// TwinCAT 3 PLC project PLC_ForTwinSAFEinTc3
// ProgramVersion: 3.1.4024.0
// libraries:
//   Tc2_EtherCAT,3.3.0.0,Beckhoff Automation GmbH
//   Tc2_MC2,3.3.2.0,Beckhoff Automation GmbH
//   Tc2_MC2_Drive,3.3.0.0,Beckhoff Automation GmbH
//   Tc2_MDP,3.3.0.0,Beckhoff Automation GmbH
//   Tc2_Standard,3.3.0.0,Beckhoff Automation GmbH
//   Tc2_System,3.3.2.0,Beckhoff Automation GmbH
//   Tc2_Utilities,3.3.1.0,Beckhoff Automation GmbH
//   Tc3_Interfaces,3.3.0.0,Beckhoff Automation GmbH
//   Tc3_Module,3.3.2.0,Beckhoff Automation GmbH
// project tree:
//   DUTs/MDP/ ST_MDP_CPU.TcDUT, ST_MDP_DiskMngmntTBL4.TcDUT, ST_MDP_DiskMngmntTBL3.TcDUT, ST_MDP_DiskMngmntTBL2.TcDUT, ST_MDP_MainboardTBL1.TcDUT, ST_MDP_DiskMngmntTBL1.TcDUT, ST_MDP_TimeTBL1.TcDUT, ST_MDP_MainboardTBL2.TcDUT (not stored), ST_MDP_MainboardTBL3.TcDUT, ST_MDP_MainboardTBL4.TcDUT, ST_MDP_NIC_Properties.TcDUT, ST_MDP_MemoryTBL1.TcDUT, ST_MDP_TimeTBL2.TcDUT
//   DUTs/Safety/ DUT_ST_InfoData.TcDUT (not stored), DUT_ST_InfoDataConnectionIn.TcDUT, DUT_ST_InfoDataConnectionOut.TcDUT, DUT_ST_InfoDataFB.TcDUT
//   / GlobalImagePool.TcGIPO (not stored), GlobalTextList.TcGTLO, PlcTask.TcTTO (not stored), Visualization Manager.TcVMO (not stored)
//   GVLs/ GVL_HMI.TcGVL, GVL_IO.TcGVL
//   POUs/Control_System_Diagnostics/ EtherCAT_Diag.TcPOU, System_Functions.TcPOU
//   POUs/ MAIN.TcPOU
//   POUs/MDP_Function_Blocks/ FB_MDP_CPU_Read.TcPOU, FB_MDP_DiskMngmnt_ReadTBL2.TcPOU, FB_MDP_DiskMngmnt_ReadTBL3.TcPOU, FB_MDP_DiskMngmnt_ReadTBL4.TcPOU, FB_MDP_Mainboard_ReadTBL1.TcPOU (not stored), FB_MDP_DiskMngmnt_ReadTBL1.TcPOU, FB_MDP_Time_ReadTBL1.TcPOU, FB_MDP_Mainboard_ReadTBL2.TcPOU, FB_MDP_Mainboard_ReadTBL3.TcPOU, FB_MDP_Mainboard_ReadTBL4.TcPOU, FB_MDP_NIC_Read.TcPOU (not stored), FB_MDP_Memory_ReadTBL1.TcPOU, FB_MDP_Time_ReadTBL2.TcPOU
//   POUs/Safety_Diagnostics/ AX5805_ADS_Reads.TcPOU, EL1904_ADS_Reads.TcPOU (not stored), EL2904_ADS_Reads.TcPOU (not stored), EL6900_ADS_Reads.TcPOU (not stored), EL6930_ADS_Reads.TcPOU, EP1908_ADS_Reads.TcPOU
//   POUs/TwinSAFE_Function_Blocks_Info/ FB_InfoAND.TcPOU (not stored), FB_InfoConnectionIn.TcPOU (not stored), FB_InfoConnectionOut.TcPOU (not stored), FB_InfoConnectionShutdown.TcPOU (not stored), FB_InfoDecoupler.TcPOU, FB_InfoEDM.TcPOU (not stored), FB_InfoEStop.TcPOU, FB_InfoMON.TcPOU, FB_InfoMuting.TcPOU, FB_InfoOperationMode.TcPOU, FB_InfoOR.TcPOU (not stored), FB_InfoRS.TcPOU, FB_InfoSafetyGroup.TcPOU, FB_InfoSR.TcPOU, FB_InfoTOF.TcPOU, FB_InfoTON.TcPOU (not stored), FB_InfoTwoHand.TcPOU (not stored)
//   VISUs/ AX5805_Specific_Diagnostics.TcVIS, AX5805_Specific_Diagnostics.TcVIS, AX5805_Specific_Diagnostics.TcVIS, EL1904_Specific_Diagnostics.TcVIS (not stored), EL1904_Specific_Diagnostics.TcVIS (not stored), EL1904_Specific_Diagnostics.TcVIS (not stored), EL2904_Specific_Diagnostics.TcVIS, EL2904_Specific_Diagnostics.TcVIS, EL2904_Specific_Diagnostics.TcVIS, EL2904_Specific_Diagnostics.TcVIS, EL6900_Specific_Diagnostics.TcVIS, EL6930_Specific_Diagnostics.TcVIS, EP1908_Specific_Diagnostics.TcVIS, EP1908_Specific_Diagnostics.TcVIS, EP1908_Specific_Diagnostics.TcVIS, EP1908_Specific_Diagnostics.TcVIS, EP6900_Specific_Diagnostics.TcVIS (not stored), EP6900_Specific_Diagnostics.TcVIS (not stored), EP6930_Specific_Diagnostics.TcVIS (not stored), EP6930_Specific_Diagnostics.TcVIS (not stored), EtherCAT_Diag1.TcVIS, EtherCAT_Diag1.TcVIS, EtherCAT_Diag1.TcVIS, EtherCAT_Diag2.TcVIS, EtherCAT_Diag2.TcVIS, EtherCAT_Diag2.TcVIS, MDP_MainboardCPUMemory.TcVIS, MDP_NicTime.TcVIS, TwinCAT_INFO.TcVIS, TwinCAT_INFO.TcVIS, TwinCAT_INFO.TcVIS, TwinSAFE.TcVIS, TwinSAFE.TcVIS, TwinSAFE.TcVIS
// real-time tasks:
//   TASK PlcTask: cycle T#1ms, priority 20, ADS port 350
// motion (NC):
//   TASK NC-Task 1 SAF: cycle T#2ms, priority 4, ADS port 501
//   TASK NC-Task 1 SVB: cycle T#10ms, priority 8, ADS port 511
//   AXIS Axis 3 (id 3)
//     OtherSettings: AllowMotionCmdToSlave=true
//     encoder EncId=1, EncType=19
//       EncPara: MaxCount=#xffffffff
//     drive DrvId=1, DrvType=16
//       DrvPara: MaxCount=#xffffffff
//         TimeComp: TaskDelayCycles=1
//     controller CtrId=1, CtrType=1
//       CtrPara: PriorControlFactor=1
//         Observer: BandWidth=20
//   AXIS Axis 4 (id 4)
//     OtherSettings: AllowMotionCmdToSlave=true
//     encoder EncId=2, EncType=19
//       EncPara: MaxCount=#xffffffff
//     drive DrvId=2, DrvType=16
//       DrvPara: MaxCount=#xffffffff
//         TimeComp: TaskDelayCycles=1
//     controller CtrId=2, CtrType=1
//       CtrPara: PriorControlFactor=1
//         Observer: BandWidth=20
// I/O:
//   DEVICE Device 1 (EtherCAT) (disabled), AmsNetId 10.12.160.29.2.1
//     Term 1 (EK1200) [EK1200-5000 EtherCAT Power supply (2A E-Bus)]
//       Term 2 (EL2004) [EL2004 4Ch. Dig. Output 24V, 0.5A]
//       Term 3 (EL1904) [EL1904, 4 Ch. Safety Input 24V, TwinSAFE]
//         modules: Module 1 (FSOES)
//       Term 4 (EL2904) [EL2904, 4 Ch. Safety Output 24V, 0.5A, TwinSAFE]
//         modules: Module 1 (FSOES), Module 2 (DO)
//       Term 5 (EL6900) [EL6900, TwinSAFE PLC]
//       Term 6 (EL1008) [EL1008 8Ch. Dig. Input 24V, 3ms]
//       Term 7 (EL2008) [EL2008 8Ch. Dig. Output 24V, 0.5A]
//       Term 8 (EL3002) [EL3002 2Ch. Ana. Input +/-10V]
//       Term 15 (EL4032) [EL4032 2Ch. Ana. Output +/-10V, 12bit]
//       Term 11 (EL7201) [EL7201 1Ch. MDP742 Servo motor output stage (50V, 4A)]
//       Term 12 (EL7201) [EL7201 1Ch. MDP742 Servo motor output stage (50V, 4A)]
//       Term 13 (EL9570) [EL9570 Buffer capacitor terminal]
//       Term 14 (EK1122) [EK1122 2 port EtherCAT junction]
//       Term 10 (EL9011) [EL9011 End Terminal]
// variable links:
//   Device 1 (EtherCAT) <-> Device 1 (EtherCAT)/Term 1 (EK1200)/Term 3 (EL1904)
//     Term 1 (EK1200)/Term 5 (EL6900)/ConnectionOutputs/Message_21 RxPDO <-> Module 1 (FSOES)/TxPDO/FSOE
//     Term 1 (EK1200)/Term 5 (EL6900)/ConnectionInputs/Message_21 TxPDO <-> Module 1 (FSOES)/RxPDO/FSOE
//   Device 1 (EtherCAT) <-> Device 1 (EtherCAT)/Term 1 (EK1200)/Term 4 (EL2904)
//     Term 1 (EK1200)/Term 5 (EL6900)/ConnectionInputs/Message_22 TxPDO <-> Module 1 (FSOES)/RxPDO/FSOE
//   Device 1 (EtherCAT) <-> Device 1 (EtherCAT)/Term 1 (EK1200)/Term 5 (EL6900)
//     Term 1 (EK1200)/Term 4 (EL2904)/Module 1 (FSOES)/TxPDO/FSOE <-> ConnectionOutputs/Message_22 RxPDO
//   NC-Task 1 SAF/Axes/Axis 3 <-> Device 1 (EtherCAT)/Term 1 (EK1200)/Term 11 (EL7201)
//     Enc/Inputs/In/nDataIn1 <-> FB Position/Position
//     Drive/Inputs/In/nState1 <-> DRV Statusword/Statusword
//     Enc/Inputs/In/nDcInputTime <-> InfoData/DcInputShift
//     Drive/Inputs/In/nDcOutputTime <-> InfoData/DcOutputShift
//     Drive/Outputs/Out/nCtrl1 <-> DRV Controlword/Controlword
//     Drive/Outputs/Out/nDataOut2 <-> DRV Target velocity/Target velocity
//     Drive/Inputs/In/nState2 <-> DRV Statusword/Statusword @bit 8
//     Drive/Outputs/Out/nCtrl2 <-> DRV Controlword/Controlword @bit 8
//   NC-Task 1 SAF/Axes/Axis 4 <-> Device 1 (EtherCAT)/Term 1 (EK1200)/Term 12 (EL7201)
//     Drive/Outputs/Out/nDataOut2 <-> DRV Target velocity/Target velocity
//     Drive/Outputs/Out/nCtrl2 <-> DRV Controlword/Controlword @bit 8
//     Enc/Inputs/In/nDcInputTime <-> InfoData/DcInputShift
//     Enc/Inputs/In/nDataIn1 <-> FB Position/Position
//     Drive/Inputs/In/nState1 <-> DRV Statusword/Statusword
//     Drive/Inputs/In/nState2 <-> DRV Statusword/Statusword @bit 8
//     Drive/Inputs/In/nDcOutputTime <-> InfoData/DcOutputShift
//     Drive/Outputs/Out/nCtrl1 <-> DRV Controlword/Controlword
//   PLC_ForTwinSAFEinTc3/PLC_ForTwinSAFEinTc3 Instance <-> Device 1 (EtherCAT)
//     PlcTask Inputs/GVL_IO.g_wStateMaster <-> Inputs/DevState
//   PLC_ForTwinSAFEinTc3/PLC_ForTwinSAFEinTc3 Instance <-> Device 1 (EtherCAT)/Term 1 (EK1200)/Term 11 (EL7201)
//     PlcTask Inputs/GVL_IO.g_stEL7201_1EcSlaveState <-> InfoData/State
//     PlcTask Inputs/GVL_IO.g_wStateEL7201_1 <-> InfoData/State
//   PLC_ForTwinSAFEinTc3/PLC_ForTwinSAFEinTc3 Instance <-> Device 1 (EtherCAT)/Term 1 (EK1200)/Term 12 (EL7201)
//     PlcTask Inputs/GVL_IO.g_stEL7201_2EcSlaveState <-> InfoData/State
//     PlcTask Inputs/GVL_IO.g_wStateEL7201_2 <-> InfoData/State
//   PLC_ForTwinSAFEinTc3/PLC_ForTwinSAFEinTc3 Instance <-> Device 1 (EtherCAT)/Term 1 (EK1200)/Term 14 (EK1122)
//     PlcTask Inputs/GVL_IO.g_stEK1122_EcSlaveState <-> InfoData/State
//     PlcTask Inputs/GVL_IO.g_wStateEK1122 <-> InfoData/State
//   PLC_ForTwinSAFEinTc3/PLC_ForTwinSAFEinTc3 Instance <-> Device 1 (EtherCAT)/Term 1 (EK1200)/Term 15 (EL4032)
//     PlcTask Inputs/GVL_IO.g_stEL4032EcSlaveState <-> InfoData/State
//     PlcTask Inputs/GVL_IO.g_wStateEL4032 <-> InfoData/State
//   PLC_ForTwinSAFEinTc3/PLC_ForTwinSAFEinTc3 Instance <-> Device 1 (EtherCAT)/Term 1 (EK1200)/Term 2 (EL2004)
//     PlcTask Outputs/GVL_IO.g_xOutput1 <-> Channel 1/Output
//     PlcTask Inputs/GVL_IO.g_wStateEL2004 <-> InfoData/State
//     PlcTask Inputs/GVL_IO.g_stEL2004EcSlaveState <-> InfoData/State
//   PLC_ForTwinSAFEinTc3/PLC_ForTwinSAFEinTc3 Instance <-> Device 1 (EtherCAT)/Term 1 (EK1200)/Term 3 (EL1904)
//     PlcTask Inputs/GVL_IO.g_stEL1904EcSlaveState <-> InfoData/State
//     PlcTask Inputs/GVL_IO.g_wStateEL1904 <-> InfoData/State
//   PLC_ForTwinSAFEinTc3/PLC_ForTwinSAFEinTc3 Instance <-> Device 1 (EtherCAT)/Term 1 (EK1200)/Term 4 (EL2904)
//     PlcTask Inputs/GVL_IO.g_wStateEL2904 <-> InfoData/State
//     PlcTask Inputs/GVL_IO.g_stEL2904EcSlaveState <-> InfoData/State
//   PLC_ForTwinSAFEinTc3/PLC_ForTwinSAFEinTc3 Instance <-> Device 1 (EtherCAT)/Term 1 (EK1200)/Term 5 (EL6900)
//     PlcTask Inputs/GVL_IO.g_xTS_SafetyGroup1_COMerror <-> StandardInputs/Standard Out Var 2
//     PlcTask Outputs/GVL_IO.g_xTS_ErrAck <-> StandardOutputs/Standard In Var 1
//     PlcTask Inputs/GVL_IO.g_xTS_SafetyGroup1_FBerror <-> StandardInputs/Standard Out Var 3
//     PlcTask Inputs/GVL_IO.g_xTS_EDM_Error <-> StandardInputs/Standard Out Var 9
//     PlcTask Inputs/GVL_IO.g_stEL6900EcSlaveState <-> InfoData/State
//     PlcTask Inputs/GVL_IO.g_xTS_EStop_Error <-> StandardInputs/Standard Out Var 5
//     PlcTask Inputs/GVL_IO.g_uiTS_ProjectCRC <-> Device Info Data/Project CRC
//     PlcTask Inputs/GVL_IO.g_stTS_InfoGroup1/usiMapDiag <-> TwinSAFE Group Info Data/TwinSafeGroup1 Info Data/Diag
//     PlcTask Inputs/GVL_IO.g_stTS_InfoConnection1/usiMapState <-> Connection Info Data/Message_21 Info Data/State
//     PlcTask Inputs/GVL_IO.g_stTS_InfoConnection2/usiMapState <-> Connection Info Data/Message_22 Info Data/State
//     PlcTask Inputs/GVL_IO.g_stTS_InfoAND1/uiMapDiag <-> Function Block Info Data/TwinSafeGroup1.Network1.FBAnd1 Info Data/Diag
//     PlcTask Inputs/GVL_IO.g_stTS_InfoAND2/uiMapDiag <-> Function Block Info Data/TwinSafeGroup1.Network1.FBAnd2 Info Data/Diag
//     PlcTask Inputs/GVL_IO.g_stTS_InfoConnection1/byInputSignals <-> Connection Info Data/Message_21 Info Data/Input Safe Data Byte 0
//     PlcTask Inputs/GVL_IO.g_wStateEL6900 <-> InfoData/State
//     PlcTask Inputs/GVL_IO.g_stTS_InfoEStop1/uiMapDiag <-> Function Block Info Data/TwinSafeGroup1.Network1.FBEstop1 Info Data/Diag
//     PlcTask Inputs/GVL_IO.g_stTS_InfoConnection2/byOutputSignals <-> Connection Info Data/Message_22 Info Data/Output Safe Data Byte 0
//     PlcTask Inputs/GVL_IO.g_stTS_InfoEDM/uiMapDiag <-> Function Block Info Data/TwinSafeGroup1.Network1.FBEdm1 Info Data/Diag
//     PlcTask Inputs/GVL_IO.g_stTS_InfoAND1/usiMapState <-> Function Block Info Data/TwinSafeGroup1.Network1.FBAnd1 Info Data/State
//     PlcTask Inputs/GVL_IO.g_stTS_InfoAND2/usiMapState <-> Function Block Info Data/TwinSafeGroup1.Network1.FBAnd2 Info Data/State
//     PlcTask Inputs/GVL_IO.g_stTS_InfoTON/uiMapDiag <-> Function Block Info Data/TwinSafeGroup1.Network1.FBTon1 Info Data/Diag
//     PlcTask Inputs/GVL_IO.g_udiTS_SerialNumber <-> Device Info Data/Serial Number
//     PlcTask Inputs/GVL_IO.g_stTS_InfoTOF/uiMapDiag <-> Function Block Info Data/TwinSafeGroup1.Network1.FBTof1 Info Data/Diag
//     PlcTask Inputs/GVL_IO.g_stTS_InfoConnection1/usiMapDiag <-> Connection Info Data/Message_21 Info Data/Diag
//     PlcTask Inputs/GVL_IO.g_stTS_InfoConnection2/usiMapDiag <-> Connection Info Data/Message_22 Info Data/Diag
//     PlcTask Inputs/GVL_IO.g_stTS_InfoTOF/usiMapState <-> Function Block Info Data/TwinSafeGroup1.Network1.FBTof1 Info Data/State
//     PlcTask Inputs/GVL_IO.g_xTS_EStop_OFF_Delay_Complete <-> StandardInputs/Standard Out Var 8
//     PlcTask Inputs/GVL_IO.g_xTS_EStop_Complete <-> StandardInputs/Standard Out Var 6
//     PlcTask Outputs/GVL_IO.g_xTS_EStop_Reset <-> StandardOutputs/Standard In Var 12
//     PlcTask Inputs/GVL_IO.g_xTS_EStop_ON_Delay_Complete <-> StandardInputs/Standard Out Var 7
//     PlcTask Inputs/GVL_IO.g_stTS_InfoGroup1/usiMapState <-> TwinSAFE Group Info Data/TwinSafeGroup1 Info Data/State
//     PlcTask Inputs/GVL_IO.g_stTS_InfoEStop1/usiMapState <-> Function Block Info Data/TwinSafeGroup1.Network1.FBEstop1 Info Data/State
//     PlcTask Inputs/GVL_IO.g_stTS_InfoEDM/usiMapState <-> Function Block Info Data/TwinSafeGroup1.Network1.FBEdm1 Info Data/State
//     PlcTask Inputs/GVL_IO.g_stTS_InfoTON/usiMapState <-> Function Block Info Data/TwinSafeGroup1.Network1.FBTon1 Info Data/State
//   PLC_ForTwinSAFEinTc3/PLC_ForTwinSAFEinTc3 Instance <-> Device 1 (EtherCAT)/Term 1 (EK1200)/Term 6 (EL1008)
//     PlcTask Inputs/GVL_IO.g_wStateEL1008 <-> InfoData/State
//     PlcTask Inputs/GVL_IO.g_stEL1008EcSlaveState <-> InfoData/State
//   PLC_ForTwinSAFEinTc3/PLC_ForTwinSAFEinTc3 Instance <-> Device 1 (EtherCAT)/Term 1 (EK1200)/Term 7 (EL2008)
//     PlcTask Inputs/GVL_IO.g_stEL2008EcSlaveState <-> InfoData/State
//     PlcTask Inputs/GVL_IO.g_wStateEL2008 <-> InfoData/State
//   PLC_ForTwinSAFEinTc3/PLC_ForTwinSAFEinTc3 Instance <-> Device 1 (EtherCAT)/Term 1 (EK1200)/Term 8 (EL3002)
//     PlcTask Inputs/GVL_IO.g_wStateEL3002 <-> InfoData/State
//     PlcTask Inputs/GVL_IO.g_stEL3002EcSlaveState <-> InfoData/State

// ---- DUTs/MDP/ST_MDP_CPU.TcDUT
TYPE ST_MDP_CPU :
STRUCT
	uiLen			:UINT;			// Length
	udiCPUfrequency	:UDINT;			// CPU Frequency in MHz
	uiCPUusage		:UINT;			// Current CPU Usage [%]
	iCPUtemp 		:INT;			// Current CPU temperature in DegC
END_STRUCT
END_TYPE

// ---- DUTs/MDP/ST_MDP_DiskMngmntTBL4.TcDUT
TYPE ST_MDP_DiskMngmntTBL4 :
STRUCT
	uiLen				:UINT;	// Length
	udiDriveType1		:UDINT;	// DRV_UNKNOWN = 0, DRV_FIXED = 1, DRV_REMOVABLE = 2, DRV_CDROM = 4 
	udiDriveType2		:UDINT;	// DRV_UNKNOWN = 0, DRV_FIXED = 1, DRV_REMOVABLE = 2, DRV_CDROM = 4 
	udiDriveType3		:UDINT;	// DRV_UNKNOWN = 0, DRV_FIXED = 1, DRV_REMOVABLE = 2, DRV_CDROM = 4 
	udiDriveType4		:UDINT;	// DRV_UNKNOWN = 0, DRV_FIXED = 1, DRV_REMOVABLE = 2, DRV_CDROM = 4 
	udiDriveType5		:UDINT;	// DRV_UNKNOWN = 0, DRV_FIXED = 1, DRV_REMOVABLE = 2, DRV_CDROM = 4 
	udiDriveType6		:UDINT;	// DRV_UNKNOWN = 0, DRV_FIXED = 1, DRV_REMOVABLE = 2, DRV_CDROM = 4 
END_STRUCT
END_TYPE

// ---- DUTs/MDP/ST_MDP_DiskMngmntTBL3.TcDUT
TYPE ST_MDP_DiskMngmntTBL3 :
STRUCT
	uiLen				:UINT;			// Length
	sFileSystemName1	:T_MaxSTRING;	// File System Name
	sFileSystemName2	:T_MaxSTRING;	// File System Name
	sFileSystemName3	:T_MaxSTRING;	// File System Name
	sFileSystemName4	:T_MaxSTRING;	// File System Name
	sFileSystemName5	:T_MaxSTRING;	// File System Name
	sFileSystemName6	:T_MaxSTRING;	// File System Name
END_STRUCT
END_TYPE

// ---- DUTs/MDP/ST_MDP_DiskMngmntTBL2.TcDUT
TYPE ST_MDP_DiskMngmntTBL2 :
STRUCT
	uiLen				:UINT;			// Length
	sVolumeLabel1		:T_MaxSTRING;	// Volume Label
	sVolumeLabel2		:T_MaxSTRING;	// Volume Label
	sVolumeLabel3		:T_MaxSTRING;	// Volume Label
	sVolumeLabel4		:T_MaxSTRING;	// Volume Label
	sVolumeLabel5		:T_MaxSTRING;	// Volume Label
	sVolumeLabel6		:T_MaxSTRING;	// Volume Label
END_STRUCT
END_TYPE

// ---- DUTs/MDP/ST_MDP_MainboardTBL1.TcDUT
TYPE ST_MDP_MainboardTBL1 :
STRUCT
	uiLen					:UINT;			// Length
	sMainboardType			:T_MaxSTRING;	// CX model
	sMainboardSN			:T_MaxSTRING;	// CX Serial number
	sMainboardProdDate		:T_MaxSTRING;	// CX production date
	udiMainboardBootCount	:UDINT;			// Number of times this CX has been booted
	udiMainboardOperTime	:UDINT;			// Number of Minutes this CX has been in operation
	diMainboardMinTemp		:DINT;			// CX lowest operating temperature monitored
	diMainboardMaxTemp		:DINT;			// CX highest operating temperature monitored
	diMainboardMinVolt		:DINT;			// CX lowest input voltage monitored in mV - 5000 is Nominal value
	diMainboardMaxVolt		:DINT;			// CX highest input voltage monitored in mV - 5000 is Nominal value
	iMainboardActualTemp	:INT;			// CX current actual temperature
END_STRUCT
END_TYPE

// ---- DUTs/MDP/ST_MDP_DiskMngmntTBL1.TcDUT
TYPE ST_MDP_DiskMngmntTBL1 :
STRUCT
	uiLen				:UINT;			// Length
	sDriveLetter1		:STRING(8);		// Drive Letter
	sDriveLetter2		:STRING(8);		// Drive Letter
	sDriveLetter3		:STRING(8);		// Drive Letter
	sDriveLetter4		:STRING(8);		// Drive Letter
	sDriveLetter5		:STRING(8);		// Drive Letter
	sDriveLetter6		:STRING(8);		// Drive Letter
END_STRUCT
END_TYPE

// ---- DUTs/MDP/ST_MDP_TimeTBL1.TcDUT
TYPE ST_MDP_TimeTBL1 :
STRUCT
	uiLen					:UINT;			// Length
	sSNTP_Server			:STRING(255);	// SNTP Server
	udiSNTP_Refresh			:UDINT;			// SNTP Refresh in Seconds
	udiSec_Since_1_1_1970	:UDINT;			// Seconds since midnight January 1, 1970
	sDateTime_Presentation	:T_MaxSTRING;	// Textual DateTime presentation (ISO 8601) YYYY-MM-DDThh:mm:ss.sTZD
	uiTimezone				:UINT;			// Timezone
END_STRUCT
END_TYPE

// ---- DUTs/MDP/ST_MDP_MainboardTBL3.TcDUT
TYPE ST_MDP_MainboardTBL3 :
STRUCT
	uiLen					:UINT;				// Length *)
	sMainboard1p05v			:STRING;			// Nominal voltage of 1.05 volt in power supply - mV
	sMainboardVccCore		:STRING;			// Nominal voltage of Vcc Core in processor - mV
	sMainboard5v			:STRING;			// Nominal voltage of 5 volt in power supply - mV
	sMainboard12v			:STRING;			// Nominal voltage of 12 volt in power supply - mV
	sMainboardVBatt			:STRING;			// Nominal voltage of 3 volt Battery - mV
	sMainboardPwrCtrlVcc	:STRING;			// Nominal voltage of 5 volt in UNKNOWN - mV
	sMainboardCX2100_5v		:STRING;			// Nominal voltage of 5 volt supply in CX2100 - mV
	sMainboardCX2100_12v	:STRING;			// Nominal voltage of 12 volt supply in CX2100 - mV
	sMainboardCX2100_24v	:STRING;			// Nominal voltage of 24 volt supply in CX2100 - mV
END_STRUCT
END_TYPE

// ---- DUTs/MDP/ST_MDP_MainboardTBL4.TcDUT
TYPE ST_MDP_MainboardTBL4 :
STRUCT
	uiLen					:UINT;			// Length
	iMainboard1p05v			:INT;			// Actual voltage of 1.05 volt in power supply - mV
	iMainboardVccCore		:INT;			// Actual voltage of Vcc Core in processor - mV
	iMainboard5v			:INT;			// Actual voltage of 5 volt in power supply - mV
	iMainboard12v			:INT;			// Actual voltage of 12 volt in power supply - mV
	iMainboardVBatt			:INT;			// Actual voltage of 3 volt Battery - mV
	iMainboardPwrCtrlVcc	:INT;			// Actual voltage of 5 volt in UNKNOWN - mV
	iMainboardCX2100_5v		:INT;			// Actual voltage of 5 volt supply in CX2100 - mV
	iMainboardCX2100_12v	:INT;			// Actual voltage of 12 volt supply in CX2100 - mV
	iMainboardCX2100_24v	:INT;			// Actual voltage of 24 volt supply in CX2100 - mV
END_STRUCT
END_TYPE

// ---- DUTs/MDP/ST_MDP_NIC_Properties.TcDUT
TYPE ST_MDP_NIC_Properties :
STRUCT
	uiLen			:UINT;			// Length
	sMACAddress		:T_MaxSTRING;	// MAC Address
	sIPAddress		:T_MaxSTRING;	// IPv4 Address
	sSubnetMask		:T_MaxSTRING;	// IPv4 Subnet Mask
	xDHCP			:BOOL;			// DHCP
	iReserved		:BYTE;
	sDefaultGateway	:T_MaxSTRING;	// IPv4 Default Gateway
END_STRUCT
END_TYPE

// ---- DUTs/MDP/ST_MDP_MemoryTBL1.TcDUT
TYPE ST_MDP_MemoryTBL1 :
STRUCT
	uiLen					:UINT;			// Length
	udiProgMemAllocated		:UDINT;			// Program Memory Allocated
	udiProgMemAvailable		:UDINT;			// Program Memory Available
	udiStorageMemAllocated	:UDINT;			// Storage Memory Allocated (available for Windows CE)
	udiStorageMemAvailable	:UDINT;			// Storage Memory Available (available for Windows CE)
	udiMemoryDivision		:UDINT;			// Memory Division (available for Windows CE)
END_STRUCT
END_TYPE

// ---- DUTs/MDP/ST_MDP_TimeTBL2.TcDUT
TYPE ST_MDP_TimeTBL2 :
STRUCT
	uiLen					:UINT;			// Length
	sTimezone1				:T_MaxSTRING;	// Timezone1
	sTimezone2				:T_MaxSTRING;	// Timezone2
	sTimezone3				:T_MaxSTRING;	// Timezone3
	sTimezone4				:T_MaxSTRING;	// Timezone4
	sTimezone5				:T_MaxSTRING;	// Timezone5
	sTimezone6				:T_MaxSTRING;	// Timezone6
	sTimezone7				:T_MaxSTRING;	// Timezone7
	sTimezone8				:T_MaxSTRING;	// Timezone8
	sTimezone9				:T_MaxSTRING;	// Timezone9
	sTimezone10				:T_MaxSTRING;	// Timezone10
	sTimezone11				:T_MaxSTRING;	// Timezone11
	sTimezone12				:T_MaxSTRING;	// Timezone12
	sTimezone13				:T_MaxSTRING;	// Timezone13
	sTimezone14				:T_MaxSTRING;	// Timezone14
	sTimezone15				:T_MaxSTRING;	// Timezone15
	sTimezone16				:T_MaxSTRING;	// Timezone16
	sTimezone17				:T_MaxSTRING;	// Timezone17
	sTimezone18				:T_MaxSTRING;	// Timezone18
	sTimezone19				:T_MaxSTRING;	// Timezone19
	sTimezone20				:T_MaxSTRING;	// Timezone20
	sTimezone21				:T_MaxSTRING;	// Timezone21
	sTimezone22				:T_MaxSTRING;	// Timezone22
	sTimezone23				:T_MaxSTRING;	// Timezone23
	sTimezone24				:T_MaxSTRING;	// Timezone24
	sTimezone25				:T_MaxSTRING;	// Timezone25
	sTimezone26				:T_MaxSTRING;	// Timezone26
	sTimezone27				:T_MaxSTRING;	// Timezone27
	sTimezone28				:T_MaxSTRING;	// Timezone28
	sTimezone29				:T_MaxSTRING;	// Timezone29
	sTimezone30				:T_MaxSTRING;	// Timezone30
	sTimezone31				:T_MaxSTRING;	// Timezone31
	sTimezone32				:T_MaxSTRING;	// Timezone32
	sTimezone33				:T_MaxSTRING;	// Timezone33
	sTimezone34				:T_MaxSTRING;	// Timezone34
	sTimezone35				:T_MaxSTRING;	// Timezone35
	sTimezone36				:T_MaxSTRING;	// Timezone36
	sTimezone37				:T_MaxSTRING;	// Timezone37
	sTimezone38				:T_MaxSTRING;	// Timezone38
	sTimezone39				:T_MaxSTRING;	// Timezone39
	sTimezone40				:T_MaxSTRING;	// Timezone40
	sTimezone41				:T_MaxSTRING;	// Timezone41
	sTimezone42				:T_MaxSTRING;	// Timezone42
	sTimezone43				:T_MaxSTRING;	// Timezone43
	sTimezone44				:T_MaxSTRING;	// Timezone44
	sTimezone45				:T_MaxSTRING;	// Timezone45
	sTimezone46				:T_MaxSTRING;	// Timezone46
	sTimezone47				:T_MaxSTRING;	// Timezone47
	sTimezone48				:T_MaxSTRING;	// Timezone48
	sTimezone49				:T_MaxSTRING;	// Timezone49
	sTimezone50				:T_MaxSTRING;	// Timezone50
	sTimezone51				:T_MaxSTRING;	// Timezone51
	sTimezone52				:T_MaxSTRING;	// Timezone52
	sTimezone53				:T_MaxSTRING;	// Timezone53
	sTimezone54				:T_MaxSTRING;	// Timezone54
	sTimezone55				:T_MaxSTRING;	// Timezone55
	sTimezone56				:T_MaxSTRING;	// Timezone56
	sTimezone57				:T_MaxSTRING;	// Timezone57
	sTimezone58				:T_MaxSTRING;	// Timezone58
	sTimezone59				:T_MaxSTRING;	// Timezone59
	sTimezone60				:T_MaxSTRING;	// Timezone60
	sTimezone61				:T_MaxSTRING;	// Timezone61
	sTimezone62				:T_MaxSTRING;	// Timezone62
	sTimezone63				:T_MaxSTRING;	// Timezone63
	sTimezone64				:T_MaxSTRING;	// Timezone64
	sTimezone65				:T_MaxSTRING;	// Timezone65
	sTimezone66				:T_MaxSTRING;	// Timezone66
	sTimezone67				:T_MaxSTRING;	// Timezone67
	sTimezone68				:T_MaxSTRING;	// Timezone68
	sTimezone69				:T_MaxSTRING;	// Timezone69
	sTimezone70				:T_MaxSTRING;	// Timezone70
	sTimezone71				:T_MaxSTRING;	// Timezone71
	sTimezone72				:T_MaxSTRING;	// Timezone72
	sTimezone73				:T_MaxSTRING;	// Timezone73
	sTimezone74				:T_MaxSTRING;	// Timezone74
	sTimezone75				:T_MaxSTRING;	// Timezone75
	sTimezone76				:T_MaxSTRING;	// Timezone76
	sTimezone77				:T_MaxSTRING;	// Timezone77
	sTimezone78				:T_MaxSTRING;	// Timezone78
	sTimezone79				:T_MaxSTRING;	// Timezone79
	sTimezone80				:T_MaxSTRING;	// Timezone80
	sTimezone81				:T_MaxSTRING;	// Timezone81
	sTimezone82				:T_MaxSTRING;	// Timezone82
	sTimezone83				:T_MaxSTRING;	// Timezone83
	sTimezone84				:T_MaxSTRING;	// Timezone84
	sTimezone85				:T_MaxSTRING;	// Timezone85
	sTimezone86				:T_MaxSTRING;	// Timezone86
	sTimezone87				:T_MaxSTRING;	// Timezone87
	sTimezone88				:T_MaxSTRING;	// Timezone88
	sTimezone89				:T_MaxSTRING;	// Timezone89
	sTimezone90				:T_MaxSTRING;	// Timezone90
	sTimezone91				:T_MaxSTRING;	// Timezone91
	sTimezone92				:T_MaxSTRING;	// Timezone92
	sTimezone93				:T_MaxSTRING;	// Timezone93
	sTimezone94				:T_MaxSTRING;	// Timezone94
	sTimezone95				:T_MaxSTRING;	// Timezone95
	sTimezone96				:T_MaxSTRING;	// Timezone96
	sTimezone97				:T_MaxSTRING;	// Timezone97
	sTimezone98				:T_MaxSTRING;	// Timezone98
	sTimezone99				:T_MaxSTRING;	// Timezone99
	sTimezone100			:T_MaxSTRING;	// Timezone100
	sTimezone101			:T_MaxSTRING;	// Timezone101
END_STRUCT
END_TYPE

// ---- DUTs/Safety/DUT_ST_InfoDataConnectionIn.TcDUT
TYPE DUT_ST_InfoDataConnectionIn :
STRUCT
	// Safety input connections use this structure
	usiMapState 				: 	USINT ;
	usiMapDiag  				: 	USINT ;
	byInputSignals 				: 	BYTE ;	
END_STRUCT
END_TYPE

// ---- DUTs/Safety/DUT_ST_InfoDataConnectionOut.TcDUT
TYPE DUT_ST_InfoDataConnectionOut :
STRUCT
	///  Safety output connections use this structure
	usiMapState					: 	USINT ;
	usiMapDiag					: 	USINT ;
	byOutputSignals				: 	BYTE ;
END_STRUCT
END_TYPE

// ---- DUTs/Safety/DUT_ST_InfoDataFB.TcDUT
TYPE DUT_ST_InfoDataFB :
STRUCT
	// Safety FBs use this structure
	usiMapState 		: 	USINT ;
	uiMapDiag  			: 	UINT ;	
END_STRUCT
END_TYPE

// ---- GVLs/GVL_HMI.TcGVL
VAR_GLOBAL
//		8-2-2012
// 		This Program has been supplied by Beckhoff Automation As-Is and is intended only as an example 
//		implementation. Functionality is not guaranteed. 
//	
	// TwinSAFE project CRC	
	g_uiHMI_ProjectCRC						: 	UINT ;
	g_udiHMI_SerialNumber					: 	UDINT ;	

	// Commands to TwinSAFE controller's safety  group
	g_xHMI_ErrAckPB							: 	BOOL ;
	g_xHMI_EStopResetPB						: 	BOOL ;

	// Feedback from TwinSAFE controller's safety group
	g_xHMI_SafetyGroup1_FBerrorLT			: 	BOOL ;
	g_xHMI_SafetyGroup1_COMerrorLT			: 	BOOL ;
	
	// Feedback from TwinSAFE controller's Function Blocks
	g_xHMI_EDMerrorLT						: 	BOOL ;
	g_xHMI_EStop_CompleteLT					: 	BOOL ;
	g_xHMI_EStop_errorLT					: 	BOOL ;
	g_xHMI_EStop_OFF_Delay_CompleteLT		: 	BOOL ;
	g_xHMI_EStop_ON_Delay_CompleteLT		: 	BOOL ;
	
	// Safety Group1 Info 
	g_sHMI_StatusGroup1						: 	STRING ;
	
	// Safety Connection1 Info
	g_sHMI_StateConn1						: 	STRING ;
	g_sHMI_DiagConn1						: 	STRING ;
	g_xHMI_EL1904Ch1						: 	BOOL ;
	g_xHMI_EL1904Ch2						: 	BOOL ;
	g_xHMI_EL1904Ch3						: 	BOOL ;
	g_xHMI_EL1904Ch4						: 	BOOL ;

	// Safety Connection2 Info
	g_sHMI_StateConn2						: 	STRING ;
	g_sHMI_DiagConn2						: 	STRING ;
	g_xHMI_EL2904Ch1						: 	BOOL ;
	g_xHMI_EL2904Ch2						: 	BOOL ;
	g_xHMI_EL2904Ch3						: 	BOOL ;
	g_xHMI_EL2904Ch4						: 	BOOL ;

	// Future Safety Connection Info for EP1908-0002
	g_xHMI_EP1908Ch1						: 	BOOL ;
	g_xHMI_EP1908Ch2						: 	BOOL ;	
	g_xHMI_EP1908Ch3						: 	BOOL ;
	g_xHMI_EP1908Ch4						: 	BOOL ;
	g_xHMI_EP1908Ch5						: 	BOOL ;
	g_xHMI_EP1908Ch6						: 	BOOL ;
	g_xHMI_EP1908Ch7						: 	BOOL ;	
	g_xHMI_EP1908Ch8						: 	BOOL ;
	
	// Safety AND#1 FB Info
	g_sHMI_StatusAND1						:	STRING ;

	// Safety EStop#1 FB Info
	g_sHMI_StatusEStop1						: 	STRING ;	
	g_sHMI_DiagEStop1						: 	STRING ;	

	// Safety AND#2 FB Info
	g_sHMI_StatusAND2						: 	STRING ;

	// Safety TON FB Info
	g_sHMI_StatusTON						: 	STRING ;

	// Safety TOF FB Info
	g_sHMI_StatusTOF						: 	STRING ;

	// Safety EDM FB Info
	g_sHMI_StatusEDM						: 	STRING ;
	g_sHMI_DiagEDM							: 	STRING ;

	//ADS Read Function Block Constants
	gc_sADSNetID							: 	STRING 		:= '10.12.160.29.2.1' ;
	gc_uiEL2004_EtherCATAdr					:	UINT 		:= 1001 ;
	gc_uiEL1904_EtherCATAdr					:	UINT 		:= 1002 ;
	gc_uiEL2904_EtherCATAdr					:	UINT 		:= 1003 ;
	gc_uiEL6900_EtherCATAdr					:	UINT 		:= 1004 ;
	gc_uiEL1008_EtherCATAdr					:	UINT 		:= 1005 ;
	gc_uiEL2008_EtherCATAdr					:	UINT 		:= 1006 ;
	gc_uiEL3002_EtherCATAdr					:	UINT 		:= 1007 ;
	gc_uiEL4032_EtherCATAdr					:	UINT 		:= 1008 ;
	gc_uiEL7201_1_EtherCATAdr				:	UINT 		:= 1009 ;
	gc_uiEL7201_2_EtherCATAdr				:	UINT 		:= 1010 ;
	gc_uiEK1122_EtherCATAdr					:	UINT 		:= 1011 ;
	
	//EL1904 Safety Terminal CoE Objects of Interest(via ADS Reads)
	g_dwHMI_EL1904Sn						: 	DWORD ;  //EL1904 Serial Number
	g_wHMI_EL1904DSw						: 	WORD ;   //EL1904 DIP Switch Setting
	g_sHMI_EL1904_HWvers					: 	STRING(2) ;//EL1904 Hardware Version
	g_sHMI_EL1904_FWvers					: 	STRING(2) ;	//EL1904 Firmware Version
	g_wHMI_EL1904PriMCTemp					: 	WORD ;   //EL1904 MC1 Actual Termperature In DegC
	g_wHMI_EL1904SecMCTemp					: 	WORD ;   //EL1904 MC2 Actual Termperature In DegC
	g_wHMI_EL1904SecMC_Volts				: 	LREAL ;  //EL1904 MC1 Actual Voltage (3.3v is nominal)
	g_wHMI_EL1904PriMC_Volts				: 	LREAL ;  //EL1904 MC2 Actual Voltage (3.3v is nominal)
	g_xHMI_EL1904SenT1						: 	BOOL ;   //EL1904 Sensor Test Error on CH1
	g_xHMI_EL1904SenT2						: 	BOOL ;   //EL1904 Sensor Test Error on CH2
	g_xHMI_EL1904SenT3						: 	BOOL ;   //EL1904 Sensor Test Error on CH3
	g_xHMI_EL1904SenT4						: 	BOOL ;   //EL1904 Sensor Test Error on CH4
	g_xHMI_EL1904_2CHEval_Pair1				: 	BOOL ;   //EL1904 2CH-Eval Error Pair1 (CH1 and CH2 not same value)
	g_xHMI_EL1904_2CHEval_Pair2				: 	BOOL ;   //EL1904 2CH-Eval Error Pair2 (CH3 and CH4 not same value)
	g_xHMI_EL1904_SMiPair_Pair1				: 	BOOL ;   //EL1904 Safety Mat Error Pair1 (CH1 and CH2 not same value)
	g_xHMI_EL1904_SMiPair_Pair2				: 	BOOL ;   //EL1904 Safety Mat Error Pair2 (CH3 and CH4 not same value)
	g_xHMI_EL1904_SMExtSupply_CH1			: 	BOOL ;   //EL1904 Safety Mat Error - External Supply CH1 (CH1 test pulses missing)
	g_xHMI_EL1904_SMExtSupply_CH2			: 	BOOL ;   //EL1904 Safety Mat Error - External Supply CH2 (CH2 test pulses missing)
	g_xHMI_EL1904_SMExtSupply_CH3			: 	BOOL ;   //EL1904 Safety Mat Error - External Supply CH3 (CH3 test pulses missing)
	g_xHMI_EL1904_SMExtSupply_CH4			: 	BOOL ;   //EL1904 Safety Mat Error - External Supply CH4 (CH4 test pulses missing)
	g_xHMI_EL1904_ErrClearPB				: 	BOOL ;   //EL1904 HMI Screen Errors Clear Pushbutton
	
	//EL1904 Safety Terminal FEATURES
	g_sHMI_EL1904_OperatingMode				: 	STRING ;  //EL1904 FEATURE - Operating Mode
	g_xHMI_EL1904_SensTestActive1			: 	BOOL ;	  //EL1904 FEATURE - CH1 Sensor Test Active
	g_xHMI_EL1904_SensTestActive2			: 	BOOL ;	  //EL1904 FEATURE - CH2 Sensor Test Active
	g_xHMI_EL1904_SensTestActive3			: 	BOOL ;	  //EL1904 FEATURE - CH3 Sensor Test Active
	g_xHMI_EL1904_SensTestActive4			: 	BOOL ;	  //EL1904 FEATURE - CH4 Sensor Test Active
	g_sHMI_EL1904_LogicCh1andCh2			: 	STRING ;  //EL1904 FEATURE - CH1 and CH2 Logic
	g_sHMI_EL1904_LogicCh3andCh4			: 	STRING ;  //EL1904 FEATURE - CH3 and CH4 Logic
	
	//EL2904 Safety Terminal CoE Objects of Interest(via ADS Reads)
	g_dwHMI_EL2904Sn						:	DWORD ;  //EL2904 Serial Number
	g_wHMI_EL2904DSw						: 	WORD ;   //EL2904 DIP Switch Setting
	g_sHMI_EL2904_HWvers					: 	STRING(2) ;//EL2904 Hardware Version
	g_sHMI_EL2904_FWvers					: 	STRING(2) ;//EL2904 Firmware Version
	g_wHMI_EL2904PriMCTemp					: 	WORD ;   //EL2904 MC1 Actual Termperature In DegC
	g_wHMI_EL2904SecMCTemp					: 	WORD ;   //EL2904 MC2 Actual Termperature In DegC
	g_wHMI_EL2904SecMC_Volts				: 	LREAL ;  //EL2904 MC1 Actual Voltage (3.3v is nominal)
	g_wHMI_EL2904PriMC_Volts				: 	LREAL ;  //EL2904 MC2 Actual Voltage (3.3v is nominal)
	g_xHMI_EL2904_ExtSup_CrossCirErr_Out1	: 	BOOL ;   //EL2904 ExtSupply, Cross-Circuit (No Test Pulses) Error on CH1
	g_xHMI_EL2904_ExtSup_CrossCirErr_Out2	: 	BOOL ;   //EL2904 ExtSupply, Cross-Circuit (No Test Pulses) Error on CH2
	g_xHMI_EL2904_ExtSup_CrossCirErr_Out3	: 	BOOL ;   //EL2904 ExtSupply, Cross-Circuit (No Test Pulses) Error on CH3
	g_xHMI_EL2904_ExtSup_CrossCirErr_Out4	: 	BOOL ;   //EL2904 ExtSupply, Cross-Circuit (No Test Pulses) Error on CH4
	g_xHMI_EL2904_OutLoadErr_Out1			: 	BOOL ;   //EL2904 Open Load, I<20mA, or I>500mA on CH1
	g_xHMI_EL2904_OutLoadErr_Out2			: 	BOOL ;   //EL2904 Open Load, I<20mA, or I>500mA on CH2
	g_xHMI_EL2904_OutLoadErr_Out3			: 	BOOL ;   //EL2904 Open Load, I<20mA, or I>500mA on CH3
	g_xHMI_EL2904_OutLoadErr_Out4			: 	BOOL ;   //EL2904 Open Load, I<20mA, or I>500mA on CH4
	g_xHMI_EL2904_PwrRailVoltageHi			: 	BOOL ;   //EL2904 Power Rail Voltage Went Above Spec (24VDC + 20% = 28.8v)
	g_xHMI_EL2904_PwrRailVoltageLo			: 	BOOL ;   //EL2904 Power Rail Voltage Went Below Spec (24VDC - 15% = 20.4v)
	g_xHMI_EL2904_TempErr_OTMc1				: 	BOOL ;   //EL2904 MicroController1 Too Hot (Internal temp - not an ambient temp)
	g_xHMI_EL2904_TempErr_OTMc2				: 	BOOL ;   //EL2904 MicroController2 Too Hot (Internal temp - not an ambient temp)
	g_xHMI_EL2904_TempErr_OTOutBoard		: 	BOOL ;   //EL2904 Outputs Board Too Hot (Too Much Load Current!)
	g_xHMI_EL2904_TempErr_UTMc1				: 	BOOL ;   //EL2904 MicroController1 Too Cold (Internal temp - not an ambient temp)
	g_xHMI_EL2904_TempErr_UTMc2				: 	BOOL ;   //EL2904 MicroController2 Too Cold (Internal temp - not an ambient temp)
	g_xHMI_EL2904_TempErr_UTOutBoard		: 	BOOL ;   //EL2904 Outputs Board Too Cold (Internal temp - not an ambient temp)
	g_xHMI_EL2904_TempErr_DiffOnBoard		: 	BOOL ;   //EL2904 Temp-Differences on Either MicroController (Internal temp - not an ambient temp)
	g_xHMI_EL2904_TempErr_DiffBetweenMc1Mc2	: 	BOOL ;   //EL2904 Temp-Differences Between MicroControllers (Internal temp - not an ambient temp)
	g_xHMI_EL2904_ErrClearPB				: 	BOOL ;   //EL2904 HMI Screen Errors Clear Pushbutton
	
	//EL2904 Safety Terminal FEATURES
	g_xHMI_EL2904_StandardOuts				: 	BOOL ;	//EL2904 FEATURE - Standard Outputs Active
	g_xHMI_EL2904_CurrentMeas				: 	BOOL ;	//EL2904 FEATURE - Current Measurement Active
	g_xHMI_EL2904_TestPulses				: 	BOOL ;	//EL2904 FEATURE - Test Pulses Active
	g_xHMI_EL2904_ErrAck					: 	BOOL ;	//EL2904 FEATURE - Error Acknowledge Active

	//EP1908-0002 Safety Terminal CoE Objects of Interest(via ADS Reads)
	g_dwHMI_EP1908Sn						: 	DWORD ;  //EP1908 Serial Number
	g_wHMI_EP1908DSw						: 	WORD ;   //EP1908 DIP Switch Setting
	g_sHMI_EP1908_HWvers					: 	STRING(2) ;//EP1908 Hardware Version
	g_sHMI_EP1908_FWvers					: 	STRING(2) ;//EP1908 Software Version
	g_wHMI_EP1908PriMCTemp					: 	WORD ;   //EP1908 MC1 Actual Termperature In DegC
	g_wHMI_EP1908SecMCTemp					: 	WORD ;   //EP1908 MC2 Actual Termperature In DegC
	g_wHMI_EP1908PriMC_Volts				: 	LREAL ;  //EP1908 MC1 Actual Voltage (3.3v is nominal)
	g_wHMI_EP1908SecMC_Volts				: 	LREAL ;  //EP1908 MC2 Actual Voltage (3.3v is nominal)
	g_xHMI_EP1908SenT1						: 	BOOL ;   //EP1908 Sensor Test Error on CH1
	g_xHMI_EP1908SenT2						: 	BOOL ;   //EP1908 Sensor Test Error on CH2
	g_xHMI_EP1908SenT3						: 	BOOL ;   //EP1908 Sensor Test Error on CH3
	g_xHMI_EP1908SenT4						: 	BOOL ;   //EP1908 Sensor Test Error on CH4
	g_xHMI_EP1908SenT5						: 	BOOL ;   //EP1908 Sensor Test Error on CH5
	g_xHMI_EP1908SenT6						: 	BOOL ;   //EP1908 Sensor Test Error on CH6
	g_xHMI_EP1908SenT7						: 	BOOL ;   //EP1908 Sensor Test Error on CH7
	g_xHMI_EP1908SenT8						: 	BOOL ;   //EP1908 Sensor Test Error on CH8
	g_xHMI_EP1908_2CHEval_Pair1				: 	BOOL ;   //EP1908 2CH-Eval Error Pair1 (CH1 and CH2 not same value)
	g_xHMI_EP1908_2CHEval_Pair2				: 	BOOL ;   //EP1908 2CH-Eval Error Pair2 (CH3 and CH4 not same value)
	g_xHMI_EP1908_2CHEval_Pair3				: 	BOOL ;   //EP1908 2CH-Eval Error Pair3 (CH5 and CH6 not same value)
	g_xHMI_EP1908_2CHEval_Pair4				: 	BOOL ;   //EP1908 2CH-Eval Error Pair4 (CH7 and CH8 not same value)
	g_xHMI_EP1908_SMiPair_Pair1				: 	BOOL ;   //EP1908 Safety Mat Error Pair1 (CH1 and CH2 not same value)
	g_xHMI_EP1908_SMiPair_Pair2				: 	BOOL ;   //EP1908 Safety Mat Error Pair2 (CH3 and CH4 not same value)
	g_xHMI_EP1908_SMiPair_Pair3				: 	BOOL ;   //EP1908 Safety Mat Error Pair3 (CH5 and CH6 not same value)
	g_xHMI_EP1908_SMiPair_Pair4				: 	BOOL ;   //EP1908 Safety Mat Error Pair4 (CH7 and CH8 not same value)
	g_xHMI_EP1908_SMExtSupply_CH1			: 	BOOL ;   //EP1908 Safety Mat Error - External Supply CH1 (CH1 test pulses missing)
	g_xHMI_EP1908_SMExtSupply_CH2			: 	BOOL ;   //EP1908 Safety Mat Error - External Supply CH2 (CH2 test pulses missing)
	g_xHMI_EP1908_SMExtSupply_CH3			: 	BOOL ;   //EP1908 Safety Mat Error - External Supply CH3 (CH3 test pulses missing)
	g_xHMI_EP1908_SMExtSupply_CH4			: 	BOOL ;   //EP1908 Safety Mat Error - External Supply CH4 (CH4 test pulses missing)
	g_xHMI_EP1908_SMExtSupply_CH5			: 	BOOL ;   //EP1908 Safety Mat Error - External Supply CH5 (CH5 test pulses missing)
	g_xHMI_EP1908_SMExtSupply_CH6			: 	BOOL ;   //EP1908 Safety Mat Error - External Supply CH6 (CH6 test pulses missing)
	g_xHMI_EP1908_SMExtSupply_CH7			: 	BOOL ;   //EP1908 Safety Mat Error - External Supply CH7 (CH7 test pulses missing)
	g_xHMI_EP1908_SMExtSupply_CH8			: 	BOOL ;   //EP1908 Safety Mat Error - External Supply CH8 (CH8 test pulses missing)
	g_xHMI_EP1908_FreqGT500_CH1				: 	BOOL ;   //EP1908 Speed Monitoring Error - CH1 Frequency Greater Than 500Hz
	g_xHMI_EP1908_FreqGT500_CH2				: 	BOOL ;   //EP1908 Speed Monitoring Error - CH2 Frequency Greater Than 500Hz
	g_xHMI_EP1908_FreqGT500_CH3				: 	BOOL ;   //EP1908 Speed Monitoring Error - CH3 Frequency Greater Than 500Hz
	g_xHMI_EP1908_FreqGT500_CH4				: 	BOOL ;   //EP1908 Speed Monitoring Error - CH4 Frequency Greater Than 500Hz
	g_xHMI_EP1908_FreqGT500_CH5				: 	BOOL ;   //EP1908 Speed Monitoring Error - CH5 Frequency Greater Than 500Hz
	g_xHMI_EP1908_FreqGT500_CH6				: 	BOOL ;   //EP1908 Speed Monitoring Error - CH6 Frequency Greater Than 500Hz
	g_xHMI_EP1908_FreqGT500_CH7				: 	BOOL ;   //EP1908 Speed Monitoring Error - CH7 Frequency Greater Than 500Hz
	g_xHMI_EP1908_FreqGT500_CH8				: 	BOOL ;   //EP1908 Speed Monitoring Error - CH8 Frequency Greater Than 500Hz
	g_xHMI_EP1908_BothInact_Pair1			: 	BOOL ;   //Error In Operating Mode: 2CH Sync Vel Control - Ch1/Ch2 cannot be inactive in this mode
	g_xHMI_EP1908_BothInact_Pair2			: 	BOOL ;   //Error In Operating Mode: 2CH Sync Vel Control - Ch3/Ch4 cannot be inactive in this mode
	g_xHMI_EP1908_BothInact_Pair3			: 	BOOL ;   //Error In Operating Mode: 2CH Sync Vel Control - Ch5/Ch6 cannot be inactive in this mode
	g_xHMI_EP1908_BothInact_Pair4			: 	BOOL ;   //Error In Operating Mode: 2CH Sync Vel Control - Ch7/Ch8 cannot be inactive in this mode
	g_xHMI_EP1908_UnequalFreg_Pair1			: 	BOOL ;   //For Ch1/Ch2 pair, two different motor speeds detected
	g_xHMI_EP1908_UnequalFreg_Pair2			: 	BOOL ;   //For Ch3/Ch4 pair, two different motor speeds detected
	g_xHMI_EP1908_UnequalFreg_Pair3			: 	BOOL ;   //For Ch5/Ch6 pair, two different motor speeds detected
	g_xHMI_EP1908_UnequalFreg_Pair4			: 	BOOL ;   //For Ch7/Ch8 pair, two different motor speeds detected
	g_xHMI_EP1908_ErrClearPB				: 	BOOL ;   //EP1908 HMI Screen Errors Clear Pushbutton

	//EP1908-0002 Safety module FEATURES	
	g_sHMI_EP1908_OperatingMode				: 	STRING ; // EP1908-0002 FEATURES: Operating Mode
	g_xHMI_EP1908_SensTestActive1			: 	BOOL ;   // EP1908-0002 FEATURES: Sensor Test Channel 1 Active/Inactive
	g_xHMI_EP1908_SensTestActive2			: 	BOOL ;   // EP1908-0002 FEATURES: Sensor Test Channel 2 Active/Inactive
	g_xHMI_EP1908_SensTestActive3			: 	BOOL ;   // EP1908-0002 FEATURES: Sensor Test Channel 3 Active/Inactive
	g_xHMI_EP1908_SensTestActive4			: 	BOOL ;   // EP1908-0002 FEATURES: Sensor Test Channel 4 Active/Inactive
	g_xHMI_EP1908_SensTestActive5			: 	BOOL ;   // EP1908-0002 FEATURES: Sensor Test Channel 5 Active/Inactive
	g_xHMI_EP1908_SensTestActive6			: 	BOOL ;   // EP1908-0002 FEATURES: Sensor Test Channel 6 Active/Inactive
	g_xHMI_EP1908_SensTestActive7			: 	BOOL ;   // EP1908-0002 FEATURES: Sensor Test Channel 7 Active/Inactive
	g_xHMI_EP1908_SensTestActive8			: 	BOOL ;   // EP1908-0002 FEATURES: Sensor Test Channel 8 Active/Inactive
	g_sHMI_EP1908_LogicCh1andCh2			: 	STRING ; // EP1908-0002 FEATURES: Logic of Channels 1 and 2
	g_sHMI_EP1908_LogicCh3andCh4			: 	STRING ; // EP1908-0002 FEATURES: Logic of Channels 3 and 4
	g_sHMI_EP1908_LogicCh5andCh6			: 	STRING ; // EP1908-0002 FEATURES: Logic of Channels 5 and 6
	g_sHMI_EP1908_LogicCh7andCh8			: 	STRING ; // EP1908-0002 FEATURES: Logic of Channels 7 and 8
	g_wHMI_EP1908_VelLimit1					: 	WORD ;   // EP1908-0002 FEATURES: Velocity Limit Value for Channel 1
	g_wHMI_EP1908_VelLimit2					: 	WORD ;   // EP1908-0002 FEATURES: Velocity Limit Value for Channel 2
	g_wHMI_EP1908_VelLimit3					: 	WORD ;   // EP1908-0002 FEATURES: Velocity Limit Value for Channel 3
	g_wHMI_EP1908_VelLimit4					: 	WORD ;   // EP1908-0002 FEATURES: Velocity Limit Value for Channel 4
	g_wHMI_EP1908_VelLimit5					: 	WORD ;   // EP1908-0002 FEATURES: Velocity Limit Value for Channel 5
	g_wHMI_EP1908_VelLimit6					: 	WORD ;   // EP1908-0002 FEATURES: Velocity Limit Value for Channel 6
	g_wHMI_EP1908_VelLimit7					: 	WORD ;   // EP1908-0002 FEATURES: Velocity Limit Value for Channel 7
	g_wHMI_EP1908_VelLimit8					: 	WORD ;   // EP1908-0002 FEATURES: Velocity Limit Value for Channel 8

	//General-Overall Safety I/O State (OK or ERROR)
	g_xHMI_EL6900_General_Error				:	BOOL ;   // EL6900 Logic Terminal Has Errors
	g_xHMI_EL6930_General_Error				:	BOOL ;	 // EL6930 Logic Terminal Has Errors
	g_xHMI_EL1904_General_Error				:	BOOL ;   // EL1904 Safety Input Terminal Has Errors
	g_xHMI_EP1908_General_Error				:	BOOL ;   // EP1908 Safety Input Module Has Errors
	g_xHMI_EL2904_General_Error				:	BOOL ;   // EL2904 Safety Output Terminal Has Errors
	g_xHMI_AX5805_General_Error				:	BOOL ;   // AX5805 Drive Safety Module Has Errors

	//EL6930 Safety Logic Terminal CoE Objects of Interest(via ADS Reads mostly)
	g_dwHMI_EL6930Sn						: 	DWORD ;      //EL6930 Serial Number
	g_wHMI_EL6930DSw						: 	WORD ;       //EL6930 DIP Switch Setting
	g_sHMI_EL6930_HWvers					: 	STRING(2) ;  //EL6930 Hardware Version
	g_sHMI_EL6930_FWvers					: 	STRING(2) ;  //EL6930 Software Version
	g_bHMI_EL6930_NoOfConnections			: 	BYTE ;       //EL6930 Safety Project: Number of Safety Connections
	g_bHMI_EL6930_NoOfSafetyGrps			: 	BYTE ;       //EL6930 Safety Project: Number of Safety Groups
	g_bHMI_EL6930_NoOfSafetyFBs				: 	BYTE ;       //EL6930 Safety Project: Number of Safety Function Blocks
	g_wHMI_EL6930PriMCTemp					: 	WORD ;       //EL6930 MC1 Actual Termperature In DegC
	g_wHMI_EL6930SecMCTemp					: 	WORD ;       //EL6930 MC2 Actual Termperature In DegC
	g_wHMI_EL6930PriMC_Volts				: 	LREAL ;      //EL6930 MC1 Actual Voltage (3.3v is nominal)
	g_wHMI_EL6930SecMC_Volts				: 	LREAL ;      //EL6930 MC2 Actual Voltage (3.3v is nominal)
	g_xHMI_EL6930_MaxTemp					: 	BOOL ;       //EL6930 Maximum Temperature Exceeded Error
	g_xHMI_EL6930_MinTemp					: 	BOOL ;       //EL6930 Temperature Fell Below Minimum Error
	g_xHMI_EL6930_TempDiffExceeded			: 	BOOL ;       //EL6930 Temperature Difference Between Measuring Points Exceeded Error
	g_xHMI_EL6930_MaxVccMC1					: 	BOOL ;       //EL6930 Maximum Supply Voltage for MC1 Exceeded Error
	g_xHMI_EL6930_MaxVccMC2					: 	BOOL ;       //EL6930 Maximum Supply Voltage for MC2 Exceeded Error
	g_xHMI_EL6930_MinVccMC1					: 	BOOL ;       //EL6930 Voltage Fell Below Minimum Supply Voltage for MC1 Error
	g_xHMI_EL6930_MinVccMC2					: 	BOOL ;       //EL6930 Voltage Fell Below Minimum Supply Voltage for MC2 Error
	g_xHMI_EL6930_ErrClearPB				: 	BOOL ;   	 //EL6930 HMI Screen Errors Clear Pushbutton

	//EL6900 Safety Logic Terminal CoE Objects of Interest(via ADS Reads mostly)
	g_dwHMI_EL6900Sn						: 	DWORD ;      //EL6900 Serial Number
	g_wHMI_EL6900DSw						: 	WORD ;       //EL6900 DIP Switch Setting
	g_sHMI_EL6900_HWvers					: 	STRING(2) ;  //EL6900 Hardware Version
	g_sHMI_EL6900_FWvers					: 	STRING(2) ;  //EL6900 Software Version
	g_bHMI_EL6900_NoOfConnections			: 	BYTE ;       //EL6900 Safety Project: Number of Safety Connections
	g_bHMI_EL6900_NoOfSafetyGrps			: 	BYTE ;       //EL6900 Safety Project: Number of Safety Groups
	g_bHMI_EL6900_NoOfSafetyFBs				: 	BYTE ;       //EL6900 Safety Project: Number of Safety Function Blocks
	g_wHMI_EL6900PriMCTemp					: 	WORD ;       //EL6900 MC1 Actual Termperature In DegC
	g_wHMI_EL6900SecMCTemp					: 	WORD ;       //EL6900 MC2 Actual Termperature In DegC
	g_wHMI_EL6900PriMC_Volts				: 	LREAL ;      //EL6900 MC1 Actual Voltage (3.3v is nominal)
	g_wHMI_EL6900SecMC_Volts				: 	LREAL ;      //EL6900 MC2 Actual Voltage (3.3v is nominal)
	g_xHMI_EL6900_MaxTemp					: 	BOOL ;       //EL6900 Maximum Temperature Exceeded Error
	g_xHMI_EL6900_MinTemp					: 	BOOL ;       //EL6900 Temperature Fell Below Minimum Error
	g_xHMI_EL6900_TempDiffExceeded			: 	BOOL ;       //EL6900 Temperature Difference Between Measuring Points Exceeded Error
	g_xHMI_EL6900_MaxVccMC1					: 	BOOL ;       //EL6900 Maximum Supply Voltage for MC1 Exceeded Error
	g_xHMI_EL6900_MaxVccMC2					: 	BOOL ;       //EL6900 Maximum Supply Voltage for MC2 Exceeded Error
	g_xHMI_EL6900_MinVccMC1					: 	BOOL ;       //EL6900 Voltage Fell Below Minimum Supply Voltage for MC1 Error
	g_xHMI_EL6900_MinVccMC2					: 	BOOL ;       //EL6900 Voltage Fell Below Minimum Supply Voltage for MC2 Error
	g_xHMI_EL6900_ErrClearPB				: 	BOOL ;   	 //EL6900 HMI Screen Errors Clear Pushbutton

(*	0  = TwinSAFE
	10 = EL1904_Specific_Diagnostics
	20 = EL1908_Specific_Diagnostics
	30 = EL2904_Specific_Diagnostics
	40 = EL6900_Specific_Diagnostics
	50 = EL6930_Specific_Diagnostics
	60 = AX5805_Specific_Diagnostics
	70 = EtherCAT_Diag1
	80 = EtherCAT_Diag2
	90 = TwinCAT_INFO  *)	
	g_bHMI_ScreenBeingDisplayed				:	BYTE ;		 //Current screen being displayed
	
	//AX5805 Safe Motion CoE Objects of Interest(via ADS Reads mostly)
	g_dwHMI_AX5805Sn						: 	DWORD ;     //AX5805 Serial Number
	g_wHMI_AX5805DSw						: 	WORD ;      //AX5805 DIP Switch Setting
	g_sHMI_AX5805_HWvers					: 	STRING(2) ; //AX5805 Hardware Version
	g_sHMI_AX5805_FWvers					: 	STRING(2) ; //AX5805 Software Version
	g_wHMI_AX5805PriMCTemp					: 	WORD ;      //AX5805 MC1 Actual Termperature In DegC
	g_wHMI_AX5805SecMCTemp					: 	WORD ;      //AX5805 MC2 Actual Termperature In DegC
	g_wHMI_AX5805PriMC_3p3Volts				: 	LREAL ;     //AX5805 MC1 Actual Voltage of 3.3v Nominal Supply
	g_wHMI_AX5805SecMC_3p3Volts				: 	LREAL ;     //AX5805 MC2 Actual Voltage of 3.3v Nominal Supply
	g_wHMI_AX5805PriMC_5Volts				: 	LREAL ;     //AX5805 MC1 Actual Voltage of 5.0v Nominal Supply
	g_wHMI_AX5805SecMC_5Volts				: 	LREAL ;     //AX5805 MC2 Actual Voltage of 5.0v Nominal Supply
	g_sHMI_AX5000_SafetyOption				: 	STRING ;    //AX5000 Safety Option (None, AX5801, AX5805)
	g_sHMI_AX5000_ConfigMotorCHA			: 	STRING ;    //AX5000 ChA Motor String
	g_sHMI_AX5000_ConfigMotorCHB			: 	STRING ;    //AX5000 ChB Motor String

	//EtherCAT Master Diagnostics
	g_sHMI_StateMaster						: 	STRING ;
	g_udiHMI_LostFrames						: 	UDINT ;
	g_lrHMI_FramesPerSecond					: 	LREAL ;
	g_udiHMI_LostQueuedFrames				: 	UDINT ;
	g_lrHMI_QueuedFramesPerSecond			: 	LREAL ;
	g_xHMI_CearMFStatCRCs					: 	BOOL ;
	g_xHMI_ClearMFStatFrames				: 	BOOL ;
	g_xHMI_ClearMFStatTxRxErr				:	BOOL ;
	g_dwHMI_TotalCrcErrors					: 	DWORD ;
	g_uiHMI_ConfSlaves						: 	UINT ;
	g_uiHMI_ScannedSlaves					: 	UINT ;

	//Check EtherCAT Slave EL2004
	g_sHMI_StateEL2004						:	STRING ;
	g_stHMI_EL2004EcSlaveStateBits			:	ST_EcSlaveStateBits ;
	g_iHMI_ProdCodeEL2004					: 	INT ;
	g_stHMI_EL2004CrcErrorEx				:	ST_EcCrcErrorEx ;

	//Check EtherCAT Slave EL1904
	g_sHMI_StateEL1904						:	STRING ;
	g_stHMI_EL1904EcSlaveStateBits			:	ST_EcSlaveStateBits ;
	g_iHMI_ProdCodeEL1904					: 	INT ;
	g_stHMI_EL1904CrcErrorEx				:	ST_EcCrcErrorEx ;

	//Check EtherCAT Slave EL2904
	g_sHMI_StateEL2904						:	STRING ;
	g_stHMI_EL2904EcSlaveStateBits			:	ST_EcSlaveStateBits ;
	g_iHMI_ProdCodeEL2904					: 	INT ;
	g_stHMI_EL2904CrcErrorEx				:	ST_EcCrcErrorEx ;
	
	//Check EtherCAT Slave EL6900
	g_sHMI_StateEL6900						:	STRING ;
	g_stHMI_EL6900EcSlaveStateBits			:	ST_EcSlaveStateBits ;
	g_iHMI_ProdCodeEL6900					: 	INT ;
	g_stHMI_EL6900CrcErrorEx				:	ST_EcCrcErrorEx ;
	
	//Check EtherCAT Slave EL1008
	g_sHMI_StateEL1008						:	STRING ;
	g_stHMI_EL1008EcSlaveStateBits			:	ST_EcSlaveStateBits ;
	g_iHMI_ProdCodeEL1008					: 	INT ;
	g_stHMI_EL1008CrcErrorEx				:	ST_EcCrcErrorEx ;

	//Check EtherCAT Slave EL2008
	g_sHMI_StateEL2008						:	STRING ;
	g_stHMI_EL2008EcSlaveStateBits			:	ST_EcSlaveStateBits ;
	g_iHMI_ProdCodeEL2008					: 	INT ;
	g_stHMI_EL2008CrcErrorEx				:	ST_EcCrcErrorEx ;
	
	//Check EtherCAT Slave EL3002
	g_sHMI_StateEL3002						:	STRING ;
	g_stHMI_EL3002EcSlaveStateBits			:	ST_EcSlaveStateBits ;
	g_iHMI_ProdCodeEL3002					: 	INT ;
	g_stHMI_EL3002CrcErrorEx				:	ST_EcCrcErrorEx ;

	//Check EtherCAT Slave EL4034
	g_sHMI_StateEL4032						:	STRING ;
	g_stHMI_EL4032EcSlaveStateBits			:	ST_EcSlaveStateBits ;
	g_iHMI_ProdCodeEL4032					: 	INT ;
	g_stHMI_EL4032CrcErrorEx				:	ST_EcCrcErrorEx ;	

	//Check EtherCAT Slave EL7201 #1
	g_sHMI_StateEL7201_1					:	STRING ;
	g_stHMI_EL7201_1EcSlaveStateBits		:	ST_EcSlaveStateBits ;
	g_iHMI_ProdCodeEL7201_1					: 	INT ;
	g_stHMI_EL7201_1CrcErrorEx				:	ST_EcCrcErrorEx ;	

	//Check EtherCAT Slave EL7201 #2
	g_sHMI_StateEL7201_2					:	STRING ;
	g_stHMI_EL7201_2EcSlaveStateBits		:	ST_EcSlaveStateBits ;
	g_iHMI_ProdCodeEL7201_2					: 	INT ;
	g_stHMI_EL7201_2CrcErrorEx				:	ST_EcCrcErrorEx ;	

	//Check EtherCAT Slave EK1122
	g_sHMI_StateEK1122						:	STRING ;
	g_stHMI_EK1122_EcSlaveStateBits			:	ST_EcSlaveStateBits ;
	g_iHMI_ProdCodeEK1122					: 	INT ;
	g_stHMI_EK1122_CrcErrorEx				:	ST_EcCrcErrorEx ;	

(*
	//Check EtherCAT Slave EL6930
	g_sHMI_StateEL6930						:	STRING ;
	g_stHMI_EL6930EcSlaveStateBits			:	ST_EcSlaveStateBits ;
	g_iHMI_ProdCodeEL6930					: 	INT ;
	g_stHMI_EL6930CrcErrorEx				:	ST_EcCrcErrorEx ;

	//Check EtherCAT Slave EK1110
	g_sHMI_StateEK1110						:	STRING ;
	g_stHMI_EK1110EcSlaveStateBits			:	ST_EcSlaveStateBits ;
	g_iHMI_ProdCodeEK1110					: 	INT ;
	g_stHMI_EK1110CrcErrorEx				:	ST_EcCrcErrorEx ;
	
	//Check EtherCAT Slave AX5000
	g_sHMI_StateAX5000						:	STRING ;
	g_stHMI_AX5000EcSlaveStateBits			:	ST_EcSlaveStateBits ;
	g_iHMI_ProdCodeAX5000					: 	INT ;
	g_stHMI_AX5000CrcErrorEx				:	ST_EcCrcErrorEx ;

	//Check EtherCAT Slave AX5805
	g_sHMI_StateAX5805						:	STRING ;
	g_stHMI_AX5805EcSlaveStateBits			:	ST_EcSlaveStateBits ;
	g_iHMI_ProdCodeAX5805					: 	INT ;
	g_stHMI_AX5805CrcErrorEx				:	ST_EcCrcErrorEx ;
	
	//Check EtherCAT Slave EP1908-0002
	g_sHMI_StateEP1908						:	STRING ;
	g_stHMI_EP1908EcSlaveStateBits			:	ST_EcSlaveStateBits ;
	g_iHMI_ProdCodeEP1908					: 	INT ;
	g_stHMI_EP1908CrcErrorEx				:	ST_EcCrcErrorEx ;	
*)

	//TwinCAT Computer and PLC INFO
	g_stHMI_DevIdent						: 	ST_DeviceIdentificationEx ;

(*
		TYPE ST_TcRouterStatusInfo

maxMem				Max. router memory byte size
maxMemAvail			Available router memory byte size
regPorts			Number of registered ports
regDrivers			Number of registered TwinCAT server ports
amsDebugLog			TRUE = Ams logging/debugging enabled, FALSE = Ams logging/debugging disabled *)
	g_stHMI_RouterStatusInfo				:	ST_TcRouterStatusInfo ;

(*
	TYPE PlcAppSystemInfo

TaskCnt 			The number of tasks in the actual runtime system. 
OnlineChangeCnt 	The number of online changes made since the last complete download. 
Flags 				Reserved for future use 
AdsPort   
BootDataLoaded   
OldBootData   
AppTimestamp   
KeepOutputsOnBP   
TComSrvPtr   
AppName   
ProjectName 		The name of the PLC project. *)
	g_stHMI_AppInfo: PlcAppSystemInfo;	
	
(*
	TYPE PlcTaskSystemInfo
 
CycleTime  			Cycletime set in the taskconfiguration in parts of 100ns. 
Priority 			Priority set in the task configuration. 
AdsPort   
CycleCount 			Cyclecounter. 
DcTaskTime   
LastExecTime 		Needed cycletime for the last cycle in parts of 100ns. 
FirstCycle 			The variable is TRUE in the first cycle of the task. 
CycleTimeExceeded 	The variable is TRUE if the runtime of the task exceeds the cycletime set in taskconfiguration. 
TaskName Contains 	the name of the task.  *)
	g_stHMI_PlcTaskSystemInfo				: 	PlcTaskSystemInfo ;
	g_lrHMI_PlcTaskSystemInfo_LastExecTime	: 	LREAL ;

	g_lrHMI_CPUfrequency					: 	LREAL;
	g_iHMI_CPUusage							: 	INT ;
	g_iHMI_CPUtemperature					: 	INT ;

	g_sHMI_MainboardType					: 	STRING(255) ;
	g_sHMI_MainboardSN						: 	STRING(255) ;
	g_sHMI_MainboardProdDate				: 	STRING(255) ;
	g_udiHMI_MainboardBootCount				: 	UDINT ;
	g_diHMI_MainboardMinTemp				: 	DINT ;
	g_diHMI_MainboardMaxTemp				: 	DINT ;
	g_iHMI_MainboardActualTemp				: 	INT ;
	g_bHMI_MainboardRevision				: 	BYTE ;
	g_bHMI_MainboardBiosMajVers				: 	BYTE ;
	g_bHMI_MainboardBiosMinVers				: 	BYTE ;
	g_sHMI_Mainboard1p05v					: 	STRING ;
	g_sHMI_MainboardVccCore					: 	STRING ;
	g_sHMI_Mainboard5v						: 	STRING ;
	g_sHMI_Mainboard12v						: 	STRING ;
	g_sHMI_MainboardVBatt					: 	STRING ;
	g_sHMI_MainboardPwrCtrlVcc				: 	STRING ;
	g_sHMI_MainboardCX2100_5v				: 	STRING ;
	g_sHMI_MainboardCX2100_12v				: 	STRING ;
	g_sHMI_MainboardCX2100_24v				: 	STRING ;
	g_lrHMI_MainboardMinVolt				: 	LREAL ;
	g_lrHMI_MainboardMaxVolt				: 	LREAL ;
	g_lrHMI_MainboardOperTimeHrs			: 	LREAL ;
	g_udiHMI_MainboardOperTimeDays			: 	UDINT ;
	g_lrHMI_Mainboard1p05v					: 	LREAL ;
	g_lrHMI_MainboardVccCore				: 	LREAL ;
	g_lrHMI_Mainboard5v						: 	LREAL ;
	g_lrHMI_Mainboard12v					: 	LREAL ;
	g_lrHMI_MainboardVBatt					: 	LREAL ;
	g_lrHMI_MainboardPwrCtrlVcc				: 	LREAL ;
	g_lrHMI_MainboardCX2100_5v				: 	LREAL ;
	g_lrHMI_MainboardCX2100_12v				: 	LREAL ;
	g_lrHMI_MainboardCX2100_24v				:	LREAL ;
	g_lrHMI_PlcTaskSystemInfo_CycleTime		: 	LREAL;
	
	g_sHMI_CurrentTimeZone					: 	STRING ;
	g_sHMI_SNTP_Server						: 	STRING(255) ;
	g_udiHMI_SNTP_Refresh					: 	UDINT ;
	g_lrHMI_SNTP_Refresh_Minutes			: 	LREAL ;
	g_lrHMI_Time_Since_1_1_1970				: 	LREAL ;
	g_lrHMI_Years_Since_1_1_1970			: 	LREAL ;
	g_sHMI_DateTime_Presentation			: 	STRING(255) ;
	g_uiHMI_Timezone						: 	UINT ;
	
	g_udiHMI_ProgMemAllocated				: 	UDINT ;
	g_udiHMI_ProgMemAvailable				: 	UDINT ;
	g_udiHMI_ProgMemUsed					: 	UDINT ;
	g_lrHMI_ProgMemAllocated_InGB: LREAL;
	g_lrHMI_ProgMemAvailable_InGB: LREAL;
	g_lrHMI_ProgMemUsed_InGB: LREAL;
	g_lrHMI_ProgStorAllocated_InGB: LREAL;
	g_lrHMI_ProgStorAvailable_InGB: LREAL;
	g_lrHMI_ProgStorUsed_InGB: LREAL;
	g_lrHMI_ProgStorMemDivision_InGB: LREAL;
END_VAR

// ---- GVLs/GVL_IO.TcGVL
VAR_GLOBAL
//		8-2-2012
// 		This Program has been supplied by Beckhoff Automation As-Is and is intended only as an example 
//		implementation. Functionality is not guaranteed. 
//
	//Some regular I/O just to have the EtherCAT bus running for TwinSAFE development
	g_xOutput1 AT %Q* 						: 	BOOL ;  // EL2004 CH1
	g_xOutput2 AT %Q* 						: 	BOOL ;	// EL2004 CH2
	g_xOutput3 AT %Q* 						: 	BOOL ;  // EL2004 CH3
	g_xOutput4 AT %Q* 						: 	BOOL ;  // EL2004 CH4
	
	// TwinSAFE project CRC	
	g_uiTS_ProjectCRC AT %I* 				:	UINT ;
	g_udiTS_SerialNumber AT %I* 			: 	UDINT ;
	
	// Commands to TwinSAFE controller's safety  group	
	g_xTS_ErrAck AT %Q* 					: 	BOOL ;
	g_xTS_EStop_Reset AT %Q*				: 	BOOL ;

	// Feedback from TwinSAFE controller's safety group
	g_xTS_SafetyGroup1_FBerror AT %I* 		:	BOOL ;
	g_xTS_SafetyGroup1_COMerror AT %I*		: 	BOOL ;
	
	// Feedback from TwinSAFE controller's Function Blocks
	g_xTS_EDM_Error AT %I* 					: 	BOOL ;
	g_xTS_EStop_Complete AT %I* 			: 	BOOL ;	
	g_xTS_EStop_Error AT %I* 				: 	BOOL ;
	g_xTS_EStop_OFF_Delay_Complete AT %I* 	: 	BOOL ;
	g_xTS_EStop_ON_Delay_Complete AT %I* 	: 	BOOL ;
	
	// Safety Group1 Info 
	g_stTS_InfoGroup1 AT %I* 				: 	DUT_ST_InfoData ;
	
	// Safety Connection1 Info
	g_stTS_InfoConnection1 AT %I* 			: 	DUT_ST_InfoDataConnectionIn ;

	// Safety Connection2 Info
	g_stTS_InfoConnection2 AT %I* 			: 	DUT_ST_InfoDataConnectionOut ;

	// Safety AND#1 FB Info
	g_stTS_InfoAND1 AT %I* 					: 	DUT_ST_InfoDataFB ;

	// Safety EStop#1 FB Info
	g_stTS_InfoEStop1 AT %I* 				: 	DUT_ST_InfoDataFB ;

	// Safety AND#2 FB Info
	g_stTS_InfoAND2 AT %I* 					: 	DUT_ST_InfoDataFB ;

	// Safety TON FB Info
	g_stTS_InfoTON AT %I* 					: 	DUT_ST_InfoDataFB ;

	// Safety TOF FB Info
	g_stTS_InfoTOF AT %I* 					: 	DUT_ST_InfoDataFB ;

	// Safety EDM FB Info
	g_stTS_InfoEDM AT %I* 					: 	DUT_ST_InfoDataFB ;

	//EtherCAT Master Diagnostics
	g_wStateMaster AT %I*					: 	WORD ;

	//Check EtherCAT Slave EL2004
	g_wStateEL2004 AT %I*					: 	WORD ;
	g_stEL2004EcSlaveState AT %I*			: 	ST_EcSlaveState ;
	g_xEL2004_Wc AT %I*						: 	BOOL ;

	//Check EtherCAT Slave EL1904
	g_wStateEL1904 AT %I*					: 	WORD ;
	g_stEL1904EcSlaveState AT %I*			: 	ST_EcSlaveState ;
	g_xEL1904_Wc AT %I*						: 	BOOL ;

	//Check EtherCAT Slave EL2904
	g_wStateEL2904 AT %I*					: 	WORD ;
	g_stEL2904EcSlaveState AT %I*			: 	ST_EcSlaveState ;
	g_xEL2904_Wc AT %I*						: 	BOOL ;
	
	//Check EtherCAT Slave EL6900
	g_wStateEL6900 AT %I*					: 	WORD ;
	g_stEL6900EcSlaveState AT %I*			: 	ST_EcSlaveState ;
	g_xEL6900_Wc AT %I*						: 	BOOL ;
	
	//Check EtherCAT Slave EL1008
	g_wStateEL1008 AT %I*					: 	WORD ;
	g_stEL1008EcSlaveState AT %I*			: 	ST_EcSlaveState ;
	g_xEL1008_Wc AT %I*						: 	BOOL ;

	//Check EtherCAT Slave EL2008
	g_wStateEL2008 AT %I*					: 	WORD ;
	g_stEL2008EcSlaveState AT %I*			: 	ST_EcSlaveState ;
	g_xEL2008_Wc AT %I*						: 	BOOL ;	
	
	//Check EtherCAT Slave EL3002
	g_wStateEL3002 AT %I*					: 	WORD ;
	g_stEL3002EcSlaveState AT %I*			: 	ST_EcSlaveState ;
	g_xEL3002_Wc AT %I*						: 	BOOL ;	
	
	//Check EtherCAT Slave EL4032
	g_wStateEL4032 AT %I*					: 	WORD ;
	g_stEL4032EcSlaveState AT %I*			: 	ST_EcSlaveState ;
	g_xEL4032_Wc AT %I*						: 	BOOL ;	

	//Check EtherCAT Slave EL7201 #1
	g_wStateEL7201_1 AT %I*					: 	WORD ;
	g_stEL7201_1EcSlaveState AT %I*			: 	ST_EcSlaveState ;
	g_xEL7201_1_Wc AT %I*					: 	BOOL ;

	//Check EtherCAT Slave EL7201 #2
	g_wStateEL7201_2 AT %I*					: 	WORD ;
	g_stEL7201_2EcSlaveState AT %I*			: 	ST_EcSlaveState ;
	g_xEL7201_2_Wc AT %I*					: 	BOOL ;

	//Check EtherCAT Slave EK1122
	g_wStateEK1122 AT %I*					: 	WORD ;
	g_stEK1122_EcSlaveState AT %I*			: 	ST_EcSlaveState ;
	g_xEK1122_Wc AT %I*						: 	BOOL ;
	
(*	//Check EtherCAT Slave EL6930
	g_wStateEL6930 AT %I*					: 	WORD ;
	g_stEL6930EcSlaveState AT %I*			: 	ST_EcSlaveState ;
	g_xEL6930_Wc AT %I*						: 	BOOL ;

	//Check EtherCAT Slave EK1110
	g_wStateEK1110 AT %I*					: 	WORD ;
	g_stEK1110EcSlaveState AT %I*			: 	ST_EcSlaveState ;
	g_xEK1110_Wc AT %I*						: 	BOOL ;
	
	//Check EtherCAT Slave AX5000
	g_wStateAX5000 AT %I*					: 	WORD ;
	g_stAX5000EcSlaveState AT %I*			: 	ST_EcSlaveState ;
	g_xAX5000_Wc AT %I*						: 	BOOL ;

	//Check EtherCAT Slave AX5805
	g_wStateAX5805 AT %I*					: 	WORD ;
	g_stAX5805EcSlaveState AT %I*			: 	ST_EcSlaveState ;
	g_xAX5805_Wc AT %I*						: 	BOOL ;
	
	//Check EtherCAT Slave EP1908-0002
	g_wStateEP1908 AT %I*					: 	WORD ;
	g_stEP1908EcSlaveState AT %I*			: 	ST_EcSlaveState ;
	g_xEP1908_Wc AT %I*						: 	BOOL ;  *)
END_VAR

// ---- POUs/Control_System_Diagnostics/EtherCAT_Diag.TcPOU
PROGRAM EtherCAT_Diag
//		8-2-2012
// 		This Program has been supplied by Beckhoff Automation As-Is and is intended only as an example 
//		implementation. Functionality is not guaranteed. 
//
VAR
	T1									: 		Ton ;
	xExecute							: 		BOOL ;
	tTime1								: 		TIME ;
	
	//Get EtherCAT network performance statistics
	fbEcMasterFrameStatistic			: 		FB_EcMasterFrameStatistic ;
	xMasterFrameStatistic_Busy			: 		BOOL ;
	xMasterFrameStatistic_Error			: 		BOOL ;
	udiMasterFrameStatistic_ErrId		: 		UDINT ;
	
	//Clear EtherCAT network CRC Errors
	fbEcMasterFrameStatisticClearCRC	:		FB_EcMasterFrameStatisticClearCRC ;
	xEcMFStatClearCRC_Busy				: 		BOOL ;
	xEcMFStatClearCRC_Error				: 		BOOL ;
	udiEcMFStatClearCRC_ErrId			: 		UDINT ;

	//Clear EtherCAT network Frame Errors
	fbEcMasterFrameStatisticClearFrames	:		FB_EcMasterFrameStatisticClearFrames ;
	xEcMFStatClearFrames_Busy			: 		BOOL ;
	xEcMFStatClearFrames_Error			: 		BOOL ;
	udiEcMFStatClearFrames_ErrId		: 		UDINT ;

	//Clear EtherCAT network Tx/Rx Errors
	fbEcMasterFrameStatisticClearTxRxErr:		FB_EcMasterFrameStatisticClearTxRxErr ;
	xEcMFStatClearTxRxErr_Busy			: 		BOOL ;
	xEcMFStatClearTxRxErr_Error			: 		BOOL ;
	udiEcMFStatClearTxRxErr_ErrId		: 		UDINT ;

	//Check for slave CRCs
	fbGetAllSlaveCrcErrors				: 		FB_EcGetAllSlaveCrcErrors ;
	ArrCrcErrors						:		ARRAY[1..12] OF DWORD ;
	xGetAllSlaveCrcErrors_Busy			: 		BOOL ;
	xGetAllSlaveCrcErrors_Error			: 		BOOL ;
	udiGetAllSlaveCrcErrors_ErrId		: 		UDINT ;
	uiGetAllSlavecrc					:		UINT ;
	udiTotalCrcErrors					: 		UDINT ;

	//Number of slaves configured
	fbEcGetConfSlaves					: 		FB_EcGetConfSlaves ;
	pArrEcConfSlaveInfo 				: 		ARRAY[0..10] OF ST_EcSlaveConfigData ;
	xGetConfSlaves_Busy					: 		BOOL ;
	xGetConfSlaves_Error				: 		BOOL ;
	udiGetConfSlaves_ErrId				: 		UDINT ;

	//Number of slaves found
	fbEcGetScannedSlaves				: 		FB_EcGetScannedSlaves ;
	xGetScannedSlaves_Busy				: 		BOOL ;
	xGetScannedSlaves_Error				: 		BOOL ;
	udiGetScannedSlaves_ErrId			: 		UDINT ;
	uiScannedSlaves						: 		UINT ;
	pArrEcScannedSlaveInfo				: 		ARRAY[0..10] OF ST_EcSlaveScannedData ;
	nScannedSlaves						: 		UINT ;

	//Get vendor product identification of EL2004 slave
	fbEL2004_EcGetSlaveIdentity			:		FB_EcGetSlaveIdentity ;
	xEL2004SlaveIdentity_Busy			:		BOOL ;
	xEL2004SlaveIdentity_Error			:		BOOL ;
	udiEL2004SlaveIdentity_ErrId		:		UDINT ;
	stSlaveIdentityEL2004				:		ST_EcSlaveIdentity ;
	sProdCodeEL2004						:		STRING ;
	sProdCodeEL2004_End4				:		STRING ;
	nProdCodeEL2004						:		INT ;

	//Check for specific CRC errors on the EL2004
	fbEL2004_EcGetSlaveCrcErrorEx		: 		FB_EcGetSlaveCrcErrorEx;
	xEL2004GetSlaveCrc_Busy				:		BOOL;
	xEL2004GetSlaveCrc_Error			:		BOOL;
	udiEL2004GetSlaveCrc_ErrId			:		UDINT;

	//Get vendor product identification of EL1904 slave
	fbEL1904_EcGetSlaveIdentity			:		FB_EcGetSlaveIdentity ;
	xEL1904SlaveIdentity_Busy			:		BOOL ;
	xEL1904SlaveIdentity_Error			:		BOOL ;
	udiEL1904SlaveIdentity_ErrId		:		UDINT ;
	stSlaveIdentityEL1904				:		ST_EcSlaveIdentity ;
	sProdCodeEL1904						:		STRING ;
	sProdCodeEL1904_End4				:		STRING ;
	nProdCodeEL1904						:		INT ;

	//Check for specific CRC errors on the EL1904
	fbEL1904_EcGetSlaveCrcErrorEx		: 		FB_EcGetSlaveCrcErrorEx;
	xEL1904GetSlaveCrc_Busy				:		BOOL;
	xEL1904GetSlaveCrc_Error			:		BOOL;
	udiEL1904GetSlaveCrc_ErrId			:		UDINT;

	//Get vendor product identification of EL2904 slave
	fbEL2904_EcGetSlaveIdentity			:		FB_EcGetSlaveIdentity ;
	xEL2904SlaveIdentity_Busy			:		BOOL ;
	xEL2904SlaveIdentity_Error			:		BOOL ;
	udiEL2904SlaveIdentity_ErrId		:		UDINT ;
	stSlaveIdentityEL2904				:		ST_EcSlaveIdentity ;
	sProdCodeEL2904						:		STRING ;
	sProdCodeEL2904_End4				:		STRING ;
	nProdCodeEL2904						:		INT ;

	//Check for specific CRC errors on the EL2904
	fbEL2904_EcGetSlaveCrcErrorEx		: 		FB_EcGetSlaveCrcErrorEx;
	xEL2904GetSlaveCrc_Busy				:		BOOL;
	xEL2904GetSlaveCrc_Error			:		BOOL;
	udiEL2904GetSlaveCrc_ErrId			:		UDINT;
	
	//Get vendor product identification of EL6900 slave
	fbEL6900_EcGetSlaveIdentity			:		FB_EcGetSlaveIdentity ;
	xEL6900SlaveIdentity_Busy			:		BOOL ;
	xEL6900SlaveIdentity_Error			:		BOOL ;
	udiEL6900SlaveIdentity_ErrId		:		UDINT ;
	stSlaveIdentityEL6900				:		ST_EcSlaveIdentity ;
	sProdCodeEL6900						:		STRING ;
	sProdCodeEL6900_End4				:		STRING ;
	nProdCodeEL6900						:		INT ;

	//Check for specific CRC errors on the EL6900
	fbEL6900_EcGetSlaveCrcErrorEx		: 		FB_EcGetSlaveCrcErrorEx;
	xEL6900GetSlaveCrc_Busy				:		BOOL;
	xEL6900GetSlaveCrc_Error			:		BOOL;
	udiEL6900GetSlaveCrc_ErrId			:		UDINT;
	
	//Get vendor product identification of EL1008 slave
	fbEL1008_EcGetSlaveIdentity			:		FB_EcGetSlaveIdentity ;
	xEL1008SlaveIdentity_Busy			:		BOOL ;
	xEL1008SlaveIdentity_Error			:		BOOL ;
	udiEL1008SlaveIdentity_ErrId		:		UDINT ;
	stSlaveIdentityEL1008				:		ST_EcSlaveIdentity ;
	sProdCodeEL1008						:		STRING ;
	sProdCodeEL1008_End4				:		STRING ;
	nProdCodeEL1008						:		INT ;

	//Check for specific CRC errors on the EL1008
	fbEL1008_EcGetSlaveCrcErrorEx		: 		FB_EcGetSlaveCrcErrorEx;
	xEL1008GetSlaveCrc_Busy				:		BOOL;
	xEL1008GetSlaveCrc_Error			:		BOOL;
	udiEL1008GetSlaveCrc_ErrId			:		UDINT;
	
	//Get vendor product identification of EL2008 slave
	fbEL2008_EcGetSlaveIdentity			:		FB_EcGetSlaveIdentity ;
	xEL2008SlaveIdentity_Busy			:		BOOL ;
	xEL2008SlaveIdentity_Error			:		BOOL ;
	udiEL2008SlaveIdentity_ErrId		:		UDINT ;
	stSlaveIdentityEL2008				:		ST_EcSlaveIdentity ;
	sProdCodeEL2008						:		STRING ;
	sProdCodeEL2008_End4				:		STRING ;
	nProdCodeEL2008						:		INT ;

	//Check for specific CRC errors on the EL2008
	fbEL2008_EcGetSlaveCrcErrorEx		: 		FB_EcGetSlaveCrcErrorEx;
	xEL2008GetSlaveCrc_Busy				:		BOOL;
	xEL2008GetSlaveCrc_Error			:		BOOL;
	udiEL2008GetSlaveCrc_ErrId			:		UDINT;
	
	//Get vendor product identification of EL3002 slave
	fbEL3002_EcGetSlaveIdentity			:		FB_EcGetSlaveIdentity ;
	xEL3002SlaveIdentity_Busy			:		BOOL ;
	xEL3002SlaveIdentity_Error			:		BOOL ;
	udiEL3002SlaveIdentity_ErrId		:		UDINT ;
	stSlaveIdentityEL3002				:		ST_EcSlaveIdentity ;
	sProdCodeEL3002						:		STRING ;
	sProdCodeEL3002_End4				:		STRING ;
	nProdCodeEL3002						:		INT ;

	//Check for specific CRC errors on the EL3002
	fbEL3002_EcGetSlaveCrcErrorEx		: 		FB_EcGetSlaveCrcErrorEx;
	xEL3002GetSlaveCrc_Busy				:		BOOL;
	xEL3002GetSlaveCrc_Error			:		BOOL;
	udiEL3002GetSlaveCrc_ErrId			:		UDINT;	
	
	//Get vendor product identification of EL4032 slave
	fbEL4032_EcGetSlaveIdentity			:		FB_EcGetSlaveIdentity ;
	xEL4032SlaveIdentity_Busy			:		BOOL ;
	xEL4032SlaveIdentity_Error			:		BOOL ;
	udiEL4032SlaveIdentity_ErrId		:		UDINT ;
	stSlaveIdentityEL4032 				: 		ST_EcSlaveIdentity ;
	sProdCodeEL4032						:		STRING ;
	sProdCodeEL4032_End4				:		STRING ;
	nProdCodeEL4032						:		INT ;

	//Check for specific CRC errors on the EL4032
	fbEL4032_EcGetSlaveCrcErrorEx		: 		FB_EcGetSlaveCrcErrorEx;
	xEL4032GetSlaveCrc_Busy				:		BOOL;
	xEL4032GetSlaveCrc_Error			:		BOOL;
	udiEL4032GetSlaveCrc_ErrId			:		UDINT;	

	//Get vendor product identification of EL7201 #1 slave
	fbEL7201_1_EcGetSlaveIdentity		:		FB_EcGetSlaveIdentity ;
	xEL7201_1SlaveIdentity_Busy			:		BOOL ;
	xEL7201_1SlaveIdentity_Error		:		BOOL ;
	udiEL7201_1SlaveIdentity_ErrId		:		UDINT ;
	stSlaveIdentityEL7201_1 			: 		ST_EcSlaveIdentity ;
	sProdCodeEL7201_1					:		STRING ;
	sProdCodeEL7201_1_End4				:		STRING ;
	nProdCodeEL7201_1					:		INT ;

	//Check for specific CRC errors on the EL7201 #1
	fbEL7201_1_EcGetSlaveCrcErrorEx		: 		FB_EcGetSlaveCrcErrorEx;
	xEL7201_1GetSlaveCrc_Busy			:		BOOL;
	xEL7201_1GetSlaveCrc_Error			:		BOOL;
	udiEL7201_1GetSlaveCrc_ErrId		:		UDINT;


	//Get vendor product identification of EL7201 #2 slave
	fbEL7201_2_EcGetSlaveIdentity		:		FB_EcGetSlaveIdentity ;
	xEL7201_2SlaveIdentity_Busy			:		BOOL ;
	xEL7201_2SlaveIdentity_Error		:		BOOL ;
	udiEL7201_2SlaveIdentity_ErrId		:		UDINT ;
	stSlaveIdentityEL7201_2 			: 		ST_EcSlaveIdentity ;
	sProdCodeEL7201_2					:		STRING ;
	sProdCodeEL7201_2_End4				:		STRING ;
	nProdCodeEL7201_2					:		INT ;

	//Check for specific CRC errors on the EL7201 #2
	fbEL7201_2_EcGetSlaveCrcErrorEx		: 		FB_EcGetSlaveCrcErrorEx;
	xEL7201_2GetSlaveCrc_Busy			:		BOOL;
	xEL7201_2GetSlaveCrc_Error			:		BOOL;
	udiEL7201_2GetSlaveCrc_ErrId		:		UDINT;

	//Get vendor product identification of EK1122 slave
	fbEK1122_EcGetSlaveIdentity			:		FB_EcGetSlaveIdentity ;
	xEK1122_SlaveIdentity_Busy			:		BOOL ;
	xEK1122_SlaveIdentity_Error			:		BOOL ;
	udiEK1122_SlaveIdentity_ErrId		:		UDINT ;
	stSlaveIdentityEK1122 				: 		ST_EcSlaveIdentity ;
	sProdCodeEK1122						:		STRING ;
	sProdCodeEK1122_End4				:		STRING ;
	nProdCodeEK1122						:		INT ;	

	//Check for specific CRC errors on the EK1122
	fbEK1122_EcGetSlaveCrcErrorEx		: 		FB_EcGetSlaveCrcErrorEx;
	xEK1122_GetSlaveCrc_Busy			:		BOOL;
	xEK1122_GetSlaveCrc_Error			:		BOOL;
	udiEK1122_GetSlaveCrc_ErrId			:		UDINT;

(*	
	//Get vendor product identification of EL6930 slave
	fbEL6930_EcGetSlaveIdentity			:		FB_EcGetSlaveIdentity ;
	xEL6930SlaveIdentity_Busy			:		BOOL ;
	xEL6930SlaveIdentity_Error			:		BOOL ;
	udiEL6930SlaveIdentity_ErrId		:		UDINT ;
	stSlaveIdentityEL6930				:		ST_EcSlaveIdentity ;
	sProdCodeEL6930						:		STRING ;
	sProdCodeEL6930_End4				:		STRING ;
	nProdCodeEL6930						:		INT ;

	//Check for specific CRC errors on the EL6930
	fbEL6930_EcGetSlaveCrcErrorEx		: 		FB_EcGetSlaveCrcErrorEx;
	xEL6930GetSlaveCrc_Busy				:		BOOL;
	xEL6930GetSlaveCrc_Error			:		BOOL;
	udiEL6930GetSlaveCrc_ErrId			:		UDINT;
	
	//Get vendor product identification of EK1110 slave
	fbEK1110_EcGetSlaveIdentity			:		FB_EcGetSlaveIdentity ;
	xEK1110SlaveIdentity_Busy			:		BOOL ;
	xEK1110SlaveIdentity_Error			:		BOOL ;
	udiEK1110SlaveIdentity_ErrId		:		UDINT ;
	stSlaveIdentityEK1110				:		ST_EcSlaveIdentity ;
	sProdCodeEK1110						:		STRING ;
	sProdCodeEK1110_End4				:		STRING ;
	nProdCodeEK1110						:		INT ;

	//Check for specific CRC errors on the EK1110
	fbEK1110_EcGetSlaveCrcErrorEx		: 		FB_EcGetSlaveCrcErrorEx;
	xEK1110GetSlaveCrc_Busy				:		BOOL;
	xEK1110GetSlaveCrc_Error			:		BOOL;
	udiEK1110GetSlaveCrc_ErrId			:		UDINT;
	
	//Get vendor product identification of AX5000 slave
	fbAX5000_EcGetSlaveIdentity			:		FB_EcGetSlaveIdentity ;
	xAX5000SlaveIdentity_Busy			:		BOOL ;
	xAX5000SlaveIdentity_Error			:		BOOL ;
	udiAX5000SlaveIdentity_ErrId		:		UDINT ;
	stSlaveIdentityAX5000				:		ST_EcSlaveIdentity ;
	sProdCodeAX5000						:		STRING ;
	sProdCodeAX5000_End4				:		STRING ;
	nProdCodeAX5000						:		INT ;

	//Check for specific CRC errors on the AX5000
	fbAX5000_EcGetSlaveCrcErrorEx		: 		FB_EcGetSlaveCrcErrorEx;
	xAX5000GetSlaveCrc_Busy				:		BOOL;
	xAX5000GetSlaveCrc_Error			:		BOOL;
	udiAX5000GetSlaveCrc_ErrId			:		UDINT;
	
	//Get vendor product identification of AX5805 slave
	fbAX5805_EcGetSlaveIdentity			:		FB_EcGetSlaveIdentity ;
	xAX5805SlaveIdentity_Busy			:		BOOL ;
	xAX5805SlaveIdentity_Error			:		BOOL ;
	udiAX5805SlaveIdentity_ErrId		:		UDINT ;
	stSlaveIdentityAX5805				:		ST_EcSlaveIdentity ;
	sProdCodeAX5805						:		STRING ;
	sProdCodeAX5805_End4				:		STRING ;
	nProdCodeAX5805						:		INT ;

	//Check for specific CRC errors on the AX5805
	fbAX5805_EcGetSlaveCrcErrorEx		: 		FB_EcGetSlaveCrcErrorEx;
	xAX5805GetSlaveCrc_Busy				:		BOOL;
	xAX5805GetSlaveCrc_Error			:		BOOL;
	udiAX5805GetSlaveCrc_ErrId			:		UDINT;
	
	//Get vendor product identification of EP1908-0002 slave
	fbEP1908_EcGetSlaveIdentity			:		FB_EcGetSlaveIdentity ;
	xEP1908SlaveIdentity_Busy			:		BOOL ;
	xEP1908SlaveIdentity_Error			:		BOOL ;
	udiEP1908SlaveIdentity_ErrId		:		UDINT ;
	stSlaveIdentityEP1908				:		ST_EcSlaveIdentity ;
	sProdCodeEP1908						:		STRING ;
	sProdCodeEP1908_End4				:		STRING ;
	nProdCodeEP1908						:		INT ;

	//Check for specific CRC errors on the EP1908-0002
	fbEP1908_EcGetSlaveCrcErrorEx		: 		FB_EcGetSlaveCrcErrorEx;
	xEP1908GetSlaveCrc_Busy				:		BOOL;
	xEP1908GetSlaveCrc_Error			:		BOOL;
	udiEP1908GetSlaveCrc_ErrId			:		UDINT;
*)
END_VAR

//		5-6-2013
// 		This Program has been supplied by Beckhoff Automation As-Is and is intended only as an example 
//		implementation. Functionality is not guaranteed. 
//

//EtherCAT Diagnostics

//IF (g_bHMI_ScreenBeingDisplayed = 70) OR (g_bHMI_ScreenBeingDisplayed = 80) THEN

//Get the state of the EtherCAT master and return status as a string - suppose to be for
//drives but works fine for any Beckhoff EtherCAT master
g_sHMI_StateMaster := F_ConvMasterDevStateToString(g_wStateMaster);

//Create the xExecute bit for continuous timed interval FB calls
T1(IN:= NOT xExecute, PT:= T#2S, Q=> xExecute, ET=>tTime1 );

//Get the EtherCAT Network Statistics
fbEcMasterFrameStatistic(		
							sNetId					:= 		gc_sADSNetID,
							bExecute				:= 		xExecute,
							tTimeout				:= 		T#2S,
							bBusy					=> 		xMasterFrameStatistic_Busy,
							bError					=> 		xMasterFrameStatistic_Error,
							nErrId					=> 		udiMasterFrameStatistic_ErrId,
							nLostFrames				=> 		g_udiHMI_LostFrames,
							fFramesPerSecond		=> 		g_lrHMI_FramesPerSecond,
							nLostQueuedFrames		=> 		g_udiHMI_LostQueuedFrames,
							fQueuedFramesPerSecond	=> 		g_lrHMI_QueuedFramesPerSecond );

//This FB sends the command to clear EtherCAT Network CRC errors
fbEcMasterFrameStatisticClearCRC(	
							sNetId					:= 		gc_sADSNetID,
							bExecute				:= 		g_xHMI_CearMFStatCRCs,
							tTimeout				:=  	T#2S,
							bBusy					=> 		xEcMFStatClearCRC_Busy,
							bError					=> 		xEcMFStatClearCRC_Error,
							nErrId					=> 		udiEcMFStatClearCRC_ErrId);

//This FB sends the command to clear EtherCAT Network Frame errors
fbEcMasterFrameStatisticClearFrames(	
							sNetId					:= 		gc_sADSNetID,
							bExecute				:= 		g_xHMI_ClearMFStatFrames,
							tTimeout				:= 		T#2S,
							bBusy					=> 		xEcMFStatClearFrames_Busy,
							bError					=> 		xEcMFStatClearFrames_Error,
							nErrId					=> 		udiEcMFStatClearFrames_ErrId);

//This FB sends the command to clear EtherCAT Network Tx/Rx errors
fbEcMasterFrameStatisticClearTxRxErr(	
							sNetId					:= 		gc_sADSNetID,
							nEcMasterDevID			:= 		1000,
							bExecute				:= 		g_xHMI_ClearMFStatTxRxErr,
							tTimeout				:= 		T#2S,
							bBusy					=> 		xEcMFStatClearTxRxErr_Busy,
							bError					=> 		xEcMFStatClearTxRxErr_Error,
							nErrId					=> 		udiEcMFStatClearTxRxErr_ErrId);
							
(* 
EtherCAT Network: Check for any CRC errors in ALL the slaves
This fuction is good for an overview but not to find the exact port (A, B, C, or D)
where the error is coming from on the terminal.  What this function does is get all
CRC errors for a terminal and simply sum them up as a single number for that slave. 
nSlaves returns how many slaves there are.  ArrCrcErrors is an array of numbers with
each number in the array representing each slave's crc summation.  For example crcError[1]
represents the sum of any crc errors for the first EtherCAT slave device in the network
and so on *)
fbGetAllSlaveCrcErrors(	
							sNetId					:= 		gc_sADSNetID,
							pCrcErrorBuf 			:= 		ADR(ArrCrcErrors),
							cbBufLen				:= 		SIZEOF(ArrCrcErrors),
							bExecute				:=		xExecute,
							tTimeout				:= 		T#2S,
							bBusy					=> 		xGetAllSlaveCrcErrors_Busy,
							bError					=> 		xGetAllSlaveCrcErrors_Error,
							nErrId					=> 		udiGetAllSlaveCrcErrors_ErrId,
							nSlaves					=> 		uiGetAllSlavecrc);

//You could be tricky here since the FB gives the number of slaves present and use that to loop through
//and sum up the total CRCs.  We didn't choose to do that for this example.
g_dwHMI_TotalCrcErrors := 	ArrCrcErrors[1] + ArrCrcErrors[2] + ArrCrcErrors[3] + ArrCrcErrors[4] + ArrCrcErrors[5] + ArrCrcErrors[6] +
							ArrCrcErrors[7] + ArrCrcErrors[8] ;

//How many slaves have been configured
fbEcGetConfSlaves(	
							sNetId					:= 		gc_sADSNetID,
							pArrEcConfSlaveInfo		:= 		ADR(pArrEcConfSlaveInfo),
							cbBufLen				:= 		SIZEOF(pArrEcConfSlaveInfo),
							bExecute				:= 		xExecute,
							tTimeout				:= 		T#2S,
							bBusy					=> 		xGetConfSlaves_Busy,
							bError					=> 		xGetConfSlaves_Error,
							nErrorId				=> 		udiGetConfSlaves_ErrId,
							nSlaves					=> 		g_uiHMI_ConfSlaves);

//How many slaves does the network see
fbEcGetScannedSlaves(	
							bExecute				:= 		xExecute,
							sNetId					:=  	gc_sADSNetID,
							pArrEcScannedSlaveInfo	:= 		ADR(pArrEcScannedSlaveInfo),
							cbBufLen				:= 		SIZEOF(pArrEcScannedSlaveInfo),
							tTimeout				:= 		T#2S,
							bBusy					=> 		xGetScannedSlaves_Busy,
							bError					=> 		xGetScannedSlaves_Error,
							nErrorId				=> 		udiGetScannedSlaves_ErrId,
							nSlaves					=> 		nScannedSlaves);
							
IF NOT xGetScannedSlaves_Busy THEN g_uiHMI_ScannedSlaves := nScannedSlaves ; END_IF ;

//Get the STATE of the EL2004 terminal and display as a text string
g_sHMI_StateEL2004 									:= 		F_ConvStateToString(g_wStateEL2004);

// slave device's STATE BITS  
g_stHMI_EL2004EcSlaveStateBits 						:=  	F_ConvSlaveStateToBits(g_stEL2004EcSlaveState);

fbEL2004_EcGetSlaveIdentity(		
							sNetId					:= 		gc_sADSNetID,
							nSlaveAddr				:= 		gc_uiEL2004_EtherCATAdr,
							bExecute				:= 		xExecute,
							tTimeout				:= 		T#2S,
							bBusy					=> 		xEL2004SlaveIdentity_Busy,
							bError					=> 		xEL2004SlaveIdentity_Error,
							nErrId					=> 		udiEL2004SlaveIdentity_ErrId,
							identity				=> 		stSlaveIdentityEL2004 );

sProdCodeEL2004 									:= 		F_ConvProductCodeToString(stSlaveIdentityEL2004);
//Get last 4 characters of the string
sProdCodeEL2004_End4 								:= 		RIGHT(sProdCodeEL2004, 4) ;
//Convert last 4 characters to a number
g_iHMI_ProdCodeEL2004 								:= 		STRING_TO_INT(sProdCodeEL2004_End4);

//In this function block the CRC counts for the individual counts can be decoded
fbEL2004_EcGetSlaveCrcErrorEx(	
							sNetId					:= 		gc_sADSNetID,
							nSlaveAddr				:= 		gc_uiEL2004_EtherCATAdr,
							bExecute				:= 		xExecute,
							tTimeout				:= 		T#2S,
							bBusy					=> 		xEL2004GetSlaveCrc_Busy,
							bError					=> 		xEL2004GetSlaveCrc_Error,
							nErrId					=> 		udiEL2004GetSlaveCrc_ErrId,
							crcError				=> 		g_stHMI_EL2004CrcErrorEx );

//Working Counter: Should remain Zero, If value=1 then data is bad from this device
g_xEL2004_Wc ;

//Get the STATE of the EL1904 terminal and display as a text string
g_sHMI_StateEL1904 									:= 		F_ConvStateToString(g_wStateEL1904);

// slave device's STATE BITS  
g_stHMI_EL1904EcSlaveStateBits 						:=  	F_ConvSlaveStateToBits(g_stEL1904EcSlaveState);

fbEL1904_EcGetSlaveIdentity(		
							sNetId					:= 		gc_sADSNetID,
							nSlaveAddr				:= 		gc_uiEL1904_EtherCATAdr,
							bExecute				:= 		xExecute,
							tTimeout				:= 		T#2S,
							bBusy					=> 		xEL1904SlaveIdentity_Busy,
							bError					=> 		xEL1904SlaveIdentity_Error,
							nErrId					=> 		udiEL1904SlaveIdentity_ErrId,
							identity				=> 		stSlaveIdentityEL1904 );

sProdCodeEL1904 									:= 		F_ConvProductCodeToString(stSlaveIdentityEL1904);
//Get last 4 characters of the string
sProdCodeEL1904_End4 								:= 		RIGHT(sProdCodeEL1904, 4) ;
//Convert last 4 characters to a number
g_iHMI_ProdCodeEL1904 								:= 		STRING_TO_INT(sProdCodeEL1904_End4);

//In this function block the CRC counts for the individual counts can be decoded
fbEL1904_EcGetSlaveCrcErrorEx(	
							sNetId					:= 		gc_sADSNetID,
							nSlaveAddr				:= 		gc_uiEL1904_EtherCATAdr,
							bExecute				:= 		xExecute,
							tTimeout				:= 		T#2S,
							bBusy					=> 		xEL1904GetSlaveCrc_Busy,
							bError					=> 		xEL1904GetSlaveCrc_Error,
							nErrId					=> 		udiEL1904GetSlaveCrc_ErrId,
							crcError				=> 		g_stHMI_EL1904CrcErrorEx );

//Working Counter: Should remain Zero, If value=1 then data is bad from this device
g_xEL1904_Wc ;


//Get the STATE of the EL2904 terminal and display as a text string
g_sHMI_StateEL2904 									:= 		F_ConvStateToString(g_wStateEL2904);

// slave device's STATE BITS  
g_stHMI_EL2904EcSlaveStateBits 						:=  	F_ConvSlaveStateToBits(g_stEL2904EcSlaveState);

fbEL2904_EcGetSlaveIdentity(		
							sNetId					:= 		gc_sADSNetID,
							nSlaveAddr				:= 		gc_uiEL2904_EtherCATAdr,
							bExecute				:= 		xExecute,
							tTimeout				:= 		T#2S,
							bBusy					=> 		xEL2904SlaveIdentity_Busy,
							bError					=> 		xEL2904SlaveIdentity_Error,
							nErrId					=> 		udiEL2904SlaveIdentity_ErrId,
							identity				=> 		stSlaveIdentityEL2904 );

sProdCodeEL2904 									:= 		F_ConvProductCodeToString(stSlaveIdentityEL2904);
//Get last 4 characters of the string
sProdCodeEL2904_End4 								:= 		RIGHT(sProdCodeEL2904, 4) ;
//Convert last 4 characters to a number
g_iHMI_ProdCodeEL2904 								:= 		STRING_TO_INT(sProdCodeEL2904_End4);

//In this function block the CRC counts for the individual counts can be decoded
fbEL2904_EcGetSlaveCrcErrorEx(	
							sNetId					:= 		gc_sADSNetID,
							nSlaveAddr				:= 		gc_uiEL2904_EtherCATAdr,
							bExecute				:= 		xExecute,
							tTimeout				:= 		T#2S,
							bBusy					=> 		xEL2904GetSlaveCrc_Busy,
							bError					=> 		xEL2904GetSlaveCrc_Error,
							nErrId					=> 		udiEL2904GetSlaveCrc_ErrId,
							crcError				=> 		g_stHMI_EL2904CrcErrorEx );

//Working Counter: Should remain Zero, If value=1 then data is bad from this device
g_xEL2904_Wc ;

//Get the STATE of the EL6900 terminal and display as a text string
g_sHMI_StateEL6900 									:= 		F_ConvStateToString(g_wStateEL6900);

(* 
Here's a really cool conversion function that decodes the STATE and presents the data
as every possible BOOL of information that is possible from the slave device's STATE.  
This function is very simply looking in the program but when viewed ONLINE the resulting
"premade" structure reveals all the available data bits *)
g_stHMI_EL6900EcSlaveStateBits 						:=  	F_ConvSlaveStateToBits(g_stEL6900EcSlaveState);

//This function is great for Beckhoff internal product info but it's a shame at this time
//the one thing it doens't support is the device's serial number!
fbEL6900_EcGetSlaveIdentity(		
							sNetId					:= 		gc_sADSNetID,
							nSlaveAddr				:= 		gc_uiEL6900_EtherCATAdr,
							bExecute				:= 		xExecute,
							tTimeout				:= 		T#2S,
							bBusy					=> 		xEL6900SlaveIdentity_Busy,
							bError					=> 		xEL6900SlaveIdentity_Error,
							nErrId					=> 		udiEL6900SlaveIdentity_ErrId,
							identity				=> 		stSlaveIdentityEL6900 );

(* 
While the EcGetSlaveIdentity FB didn't seem to be very worthwhile it was needed
in order to do the conversion function to convert to the product code which DOES say
the device's XML revision.  For example: EK1100-0000-0017 means f/w rev 17 for this
slave device *)
sProdCodeEL6900 									:= 		F_ConvProductCodeToString(stSlaveIdentityEL6900);

//Get last 4 characters of the string
sProdCodeEL6900_End4 								:= 		RIGHT(sProdCodeEL6900, 4) ;

//Convert last 4 characters to a number
g_iHMI_ProdCodeEL6900 								:= 		STRING_TO_INT(sProdCodeEL6900_End4);

//In this function block the CRC counts for the individual counts can be decoded
fbEL6900_EcGetSlaveCrcErrorEx(	
							sNetId					:= 		gc_sADSNetID,
							nSlaveAddr				:= 		gc_uiEL6900_EtherCATAdr,
							bExecute				:= 		xExecute,
							tTimeout				:= 		T#2S,
							bBusy					=> 		xEL6900GetSlaveCrc_Busy,
							bError					=> 		xEL6900GetSlaveCrc_Error,
							nErrId					=> 		udiEL6900GetSlaveCrc_ErrId,
							crcError				=> 		g_stHMI_EL6900CrcErrorEx );

//Working Counter: Should remain Zero, If value=1 then data is bad from this device
g_xEL6900_Wc ;


//Get the STATE of the EL1008 terminal and display as a text string
g_sHMI_StateEL1008 									:= 		F_ConvStateToString(g_wStateEL1008);

// slave device's STATE BITS  
g_stHMI_EL1008EcSlaveStateBits 						:=  	F_ConvSlaveStateToBits(g_stEL1008EcSlaveState);

fbEL1008_EcGetSlaveIdentity(		
							sNetId					:= 		gc_sADSNetID,
							nSlaveAddr				:= 		gc_uiEL1008_EtherCATAdr,
							bExecute				:= 		xExecute,
							tTimeout				:= 		T#2S,
							bBusy					=> 		xEL1008SlaveIdentity_Busy,
							bError					=> 		xEL1008SlaveIdentity_Error,
							nErrId					=> 		udiEL1008SlaveIdentity_ErrId,
							identity				=> 		stSlaveIdentityEL1008 );

sProdCodeEL1008 									:= 		F_ConvProductCodeToString(stSlaveIdentityEL1008);
//Get last 4 characters of the string
sProdCodeEL1008_End4 								:= 		RIGHT(sProdCodeEL1008, 4) ;
//Convert last 4 characters to a number
g_iHMI_ProdCodeEL1008 								:= 		STRING_TO_INT(sProdCodeEL1008_End4);

//In this function block the CRC counts for the individual counts can be decoded
fbEL1008_EcGetSlaveCrcErrorEx(	
							sNetId					:= 		gc_sADSNetID,
							nSlaveAddr				:= 		gc_uiEL1008_EtherCATAdr,
							bExecute				:= 		xExecute,
							tTimeout				:= 		T#2S,
							bBusy					=> 		xEL1008GetSlaveCrc_Busy,
							bError					=> 		xEL1008GetSlaveCrc_Error,
							nErrId					=> 		udiEL1008GetSlaveCrc_ErrId,
							crcError				=> 		g_stHMI_EL1008CrcErrorEx );

//Working Counter: Should remain Zero, If value=1 then data is bad from this device
g_xEL1008_Wc ;


//Get the STATE of the EL2008 terminal and display as a text string
g_sHMI_StateEL2008 									:= 		F_ConvStateToString(g_wStateEL2008);

// slave device's STATE BITS  
g_stHMI_EL2008EcSlaveStateBits 						:=  	F_ConvSlaveStateToBits(g_stEL2008EcSlaveState);

fbEL2008_EcGetSlaveIdentity(		
							sNetId					:= 		gc_sADSNetID,
							nSlaveAddr				:= 		gc_uiEL2008_EtherCATAdr,
							bExecute				:= 		xExecute,
							tTimeout				:= 		T#2S,
							bBusy					=> 		xEL2008SlaveIdentity_Busy,
							bError					=> 		xEL2008SlaveIdentity_Error,
							nErrId					=> 		udiEL2008SlaveIdentity_ErrId,
							identity				=> 		stSlaveIdentityEL2008 );

sProdCodeEL2008 									:= 		F_ConvProductCodeToString(stSlaveIdentityEL2008);
//Get last 4 characters of the string
sProdCodeEL2008_End4 								:= 		RIGHT(sProdCodeEL2008, 4) ;
//Convert last 4 characters to a number
g_iHMI_ProdCodeEL2008 								:= 		STRING_TO_INT(sProdCodeEL2008_End4);

//In this function block the CRC counts for the individual counts can be decoded
fbEL2008_EcGetSlaveCrcErrorEx(	
							sNetId					:= 		gc_sADSNetID,
							nSlaveAddr				:= 		gc_uiEL2008_EtherCATAdr,
							bExecute				:= 		xExecute,
							tTimeout				:= 		T#2S,
							bBusy					=> 		xEL2008GetSlaveCrc_Busy,
							bError					=> 		xEL2008GetSlaveCrc_Error,
							nErrId					=> 		udiEL2008GetSlaveCrc_ErrId,
							crcError				=> 		g_stHMI_EL2008CrcErrorEx );

//Working Counter: Should remain Zero, If value=1 then data is bad from this device
g_xEL2008_Wc ;



//Get the STATE of the EL3002 terminal and display as a text string
g_sHMI_StateEL3002 									:= 		F_ConvStateToString(g_wStateEL3002);

// slave device's STATE BITS  
g_stHMI_EL3002EcSlaveStateBits 						:=  	F_ConvSlaveStateToBits(g_stEL3002EcSlaveState);

fbEL3002_EcGetSlaveIdentity(		
							sNetId					:= 		gc_sADSNetID,
							nSlaveAddr				:= 		gc_uiEL3002_EtherCATAdr,
							bExecute				:= 		xExecute,
							tTimeout				:= 		T#2S,
							bBusy					=> 		xEL3002SlaveIdentity_Busy,
							bError					=> 		xEL3002SlaveIdentity_Error,
							nErrId					=> 		udiEL3002SlaveIdentity_ErrId,
							identity				=> 		stSlaveIdentityEL3002 );

sProdCodeEL3002 									:= 		F_ConvProductCodeToString(stSlaveIdentityEL3002);
//Get last 4 characters of the string
sProdCodeEL3002_End4 								:= 		RIGHT(sProdCodeEL3002, 4) ;
//Convert last 4 characters to a number
g_iHMI_ProdCodeEL3002 								:= 		STRING_TO_INT(sProdCodeEL3002_End4);

//In this function block the CRC counts for the individual counts can be decoded
fbEL3002_EcGetSlaveCrcErrorEx(	
							sNetId					:= 		gc_sADSNetID,
							nSlaveAddr				:= 		gc_uiEL3002_EtherCATAdr,
							bExecute				:= 		xExecute,
							tTimeout				:= 		T#2S,
							bBusy					=> 		xEL3002GetSlaveCrc_Busy,
							bError					=> 		xEL3002GetSlaveCrc_Error,
							nErrId					=> 		udiEL3002GetSlaveCrc_ErrId,
							crcError				=> 		g_stHMI_EL3002CrcErrorEx );

//Working Counter: Should remain Zero, If value=1 then data is bad from this device
g_xEL3002_Wc ;


//Get the STATE of the EL4032 terminal and display as a text string
g_sHMI_StateEL4032 									:= 		F_ConvStateToString(g_wStateEL4032);

// slave device's STATE BITS  
g_stHMI_EL4032EcSlaveStateBits 						:=  	F_ConvSlaveStateToBits(g_stEL4032EcSlaveState);

fbEL4032_EcGetSlaveIdentity(		
							sNetId					:= 		gc_sADSNetID,
							nSlaveAddr				:= 		gc_uiEL4032_EtherCATAdr,
							bExecute				:= 		xExecute,
							tTimeout				:= 		T#2S,
							bBusy					=> 		xEL4032SlaveIdentity_Busy,
							bError					=> 		xEL4032SlaveIdentity_Error,
							nErrId					=> 		udiEL4032SlaveIdentity_ErrId,
							identity				=> 		stSlaveIdentityEL4032 );

sProdCodeEL4032 									:= 		F_ConvProductCodeToString(stSlaveIdentityEL4032);
//Get last 4 characters of the string
sProdCodeEL4032_End4 								:= 		RIGHT(sProdCodeEL4032, 4) ;
//Convert last 4 characters to a number
g_iHMI_ProdCodeEL4032 								:= 		STRING_TO_INT(sProdCodeEL4032_End4);

//In this function block the CRC counts for the individual counts can be decoded
fbEL4032_EcGetSlaveCrcErrorEx(	
							sNetId					:= 		gc_sADSNetID,
							nSlaveAddr				:= 		gc_uiEL4032_EtherCATAdr,
							bExecute				:= 		xExecute,
							tTimeout				:= 		T#2S,
							bBusy					=> 		xEL4032GetSlaveCrc_Busy,
							bError					=> 		xEL4032GetSlaveCrc_Error,
							nErrId					=> 		udiEL4032GetSlaveCrc_ErrId,
							crcError				=> 		g_stHMI_EL4032CrcErrorEx );

//Working Counter: Should remain Zero, If value=1 then data is bad from this device
g_xEL4032_Wc ;

//Get the STATE of the EL7201 #1 terminal and display as a text string
g_sHMI_StateEL7201_1								:= 		F_ConvStateToString(g_wStateEL7201_1);

// slave device's STATE BITS  
g_stHMI_EL7201_1EcSlaveStateBits 					:=  	F_ConvSlaveStateToBits(g_stEL7201_1EcSlaveState);

fbEL7201_1_EcGetSlaveIdentity(		
							sNetId					:= 		gc_sADSNetID,
							nSlaveAddr				:= 		gc_uiEL7201_1_EtherCATAdr,
							bExecute				:= 		xExecute,
							tTimeout				:= 		T#2S,
							bBusy					=> 		xEL7201_1SlaveIdentity_Busy,
							bError					=> 		xEL7201_1SlaveIdentity_Error,
							nErrId					=> 		udiEL7201_1SlaveIdentity_ErrId,
							identity				=> 		stSlaveIdentityEL7201_1 );

sProdCodeEL7201_1 									:= 		F_ConvProductCodeToString(stSlaveIdentityEL7201_1);
//Get last 4 characters of the string
sProdCodeEL7201_1_End4 								:= 		RIGHT(sProdCodeEL7201_1, 4) ;
//Convert last 4 characters to a number
g_iHMI_ProdCodeEL7201_1 							:= 		STRING_TO_INT(sProdCodeEL7201_1_End4);

//In this function block the CRC counts for the individual counts can be decoded
fbEL7201_1_EcGetSlaveCrcErrorEx(	
							sNetId					:= 		gc_sADSNetID,
							nSlaveAddr				:= 		gc_uiEL7201_1_EtherCATAdr,
							bExecute				:= 		xExecute,
							tTimeout				:= 		T#2S,
							bBusy					=> 		xEL7201_1GetSlaveCrc_Busy,
							bError					=> 		xEL7201_1GetSlaveCrc_Error,
							nErrId					=> 		udiEL7201_1GetSlaveCrc_ErrId,
							crcError				=> 		g_stHMI_EL7201_1CrcErrorEx );

//Working Counter: Should remain Zero, If value=1 then data is bad from this device
g_xEL7201_1_Wc ;


//Get the STATE of the EL7201 #2 terminal and display as a text string
g_sHMI_StateEL7201_2								:= 		F_ConvStateToString(g_wStateEL7201_2);

// slave device's STATE BITS  
g_stHMI_EL7201_2EcSlaveStateBits 					:=  	F_ConvSlaveStateToBits(g_stEL7201_2EcSlaveState);

fbEL7201_2_EcGetSlaveIdentity(		
							sNetId					:= 		gc_sADSNetID,
							nSlaveAddr				:= 		gc_uiEL7201_2_EtherCATAdr,
							bExecute				:= 		xExecute,
							tTimeout				:= 		T#2S,
							bBusy					=> 		xEL7201_2SlaveIdentity_Busy,
							bError					=> 		xEL7201_2SlaveIdentity_Error,
							nErrId					=> 		udiEL7201_2SlaveIdentity_ErrId,
							identity				=> 		stSlaveIdentityEL7201_2 );

sProdCodeEL7201_2 									:= 		F_ConvProductCodeToString(stSlaveIdentityEL7201_2);
//Get last 4 characters of the string
sProdCodeEL7201_2_End4 								:= 		RIGHT(sProdCodeEL7201_2, 4) ;
//Convert last 4 characters to a number
g_iHMI_ProdCodeEL7201_2 							:= 		STRING_TO_INT(sProdCodeEL7201_2_End4);

//In this function block the CRC counts for the individual counts can be decoded
fbEL7201_2_EcGetSlaveCrcErrorEx(	
							sNetId					:= 		gc_sADSNetID,
							nSlaveAddr				:= 		gc_uiEL7201_2_EtherCATAdr,
							bExecute				:= 		xExecute,
							tTimeout				:= 		T#2S,
							bBusy					=> 		xEL7201_2GetSlaveCrc_Busy,
							bError					=> 		xEL7201_2GetSlaveCrc_Error,
							nErrId					=> 		udiEL7201_2GetSlaveCrc_ErrId,
							crcError				=> 		g_stHMI_EL7201_2CrcErrorEx );

//Working Counter: Should remain Zero, If value=1 then data is bad from this device
g_xEL7201_2_Wc ;


//Get the STATE of the EK1122 terminal and display as a text string
g_sHMI_StateEK1122								:= 		F_ConvStateToString(g_wStateEK1122);

// slave device's STATE BITS  
g_stHMI_EK1122_EcSlaveStateBits 					:=  	F_ConvSlaveStateToBits(g_stEK1122_EcSlaveState);

fbEK1122_EcGetSlaveIdentity(		
							sNetId					:= 		gc_sADSNetID,
							nSlaveAddr				:= 		gc_uiEK1122_EtherCATAdr,
							bExecute				:= 		xExecute,
							tTimeout				:= 		T#2S,
							bBusy					=> 		xEK1122_SlaveIdentity_Busy,
							bError					=> 		xEK1122_SlaveIdentity_Error,
							nErrId					=> 		udiEK1122_SlaveIdentity_ErrId,
							identity				=> 		stSlaveIdentityEK1122 );

sProdCodeEK1122 									:= 		F_ConvProductCodeToString(stSlaveIdentityEK1122);
//Get last 4 characters of the string
sProdCodeEK1122_End4 								:= 		RIGHT(sProdCodeEK1122, 4) ;
//Convert last 4 characters to a number
g_iHMI_ProdCodeEK1122 							:= 		STRING_TO_INT(sProdCodeEK1122_End4);

//In this function block the CRC counts for the individual counts can be decoded
fbEK1122_EcGetSlaveCrcErrorEx(	
							sNetId					:= 		gc_sADSNetID,
							nSlaveAddr				:= 		gc_uiEK1122_EtherCATAdr,
							bExecute				:= 		xExecute,
							tTimeout				:= 		T#2S,
							bBusy					=> 		xEK1122_GetSlaveCrc_Busy,
							bError					=> 		xEK1122_GetSlaveCrc_Error,
							nErrId					=> 		udiEK1122_GetSlaveCrc_ErrId,
							crcError				=> 		g_stHMI_EK1122_CrcErrorEx );

(*
//Get the STATE of the EL6930 terminal and display as a text string
g_sHMI_StateEL6930 									:= 		F_ConvStateToString(g_wStateEL6930);

// slave device's STATE BITS  
g_stHMI_EL6930EcSlaveStateBits 						:=  	F_ConvSlaveStateToBits(g_stEL6930EcSlaveState);

fbEL6930_EcGetSlaveIdentity(		
							sNetId					:= 		gc_sADSNetID,
							nSlaveAddr				:= 		gc_uiEL6930_EtherCATAdr,
							bExecute				:= 		xExecute,
							tTimeout				:= 		T#2S,
							bBusy					=> 		xEL6930SlaveIdentity_Busy,
							bError					=> 		xEL6930SlaveIdentity_Error,
							nErrId					=> 		udiEL6930SlaveIdentity_ErrId,
							identity				=> 		stSlaveIdentityEL6930 );

sProdCodeEL6930 									:= 		F_ConvProductCodeToString(stSlaveIdentityEL6930);
//Get last 4 characters of the string
sProdCodeEL6930_End4 								:= 		RIGHT(sProdCodeEL6930, 4) ;
//Convert last 4 characters to a number
g_iHMI_ProdCodeEL6930 								:= 		STRING_TO_INT(sProdCodeEL6930_End4);

//In this function block the CRC counts for the individual counts can be decoded
fbEL6930_EcGetSlaveCrcErrorEx(	
							sNetId					:= 		gc_sADSNetID,
							nSlaveAddr				:= 		gc_uiEL6930_EtherCATAdr,
							bExecute				:= 		xExecute,
							tTimeout				:= 		T#2S,
							bBusy					=> 		xEL6930GetSlaveCrc_Busy,
							bError					=> 		xEL6930GetSlaveCrc_Error,
							nErrId					=> 		udiEL6930GetSlaveCrc_ErrId,
							crcError				=> 		g_stHMI_EL6930CrcErrorEx );

//Working Counter: Should remain Zero, If value=1 then data is bad from this device
g_xEL6930_Wc;


//Get the STATE of the EK1110 terminal and display as a text string
g_sHMI_StateEK1110 									:= 		F_ConvStateToString(g_wStateEK1110);

// slave device's STATE BITS  
g_stHMI_EK1110EcSlaveStateBits 						:=  	F_ConvSlaveStateToBits(g_stEK1110EcSlaveState);

fbEK1110_EcGetSlaveIdentity(		
							sNetId					:= 		gc_sADSNetID,
							nSlaveAddr				:= 		gc_uiEK1110_EtherCATAdr,
							bExecute				:= 		xExecute,
							tTimeout				:= 		T#2S,
							bBusy					=> 		xEK1110SlaveIdentity_Busy,
							bError					=> 		xEK1110SlaveIdentity_Error,
							nErrId					=> 		udiEK1110SlaveIdentity_ErrId,
							identity				=> 		stSlaveIdentityEK1110 );

sProdCodeEK1110 									:= 		F_ConvProductCodeToString(stSlaveIdentityEL6930);
//Get last 4 characters of the string
sProdCodeEK1110_End4 								:= 		RIGHT(sProdCodeEK1110, 4) ;
//Convert last 4 characters to a number
g_iHMI_ProdCodeEK1110 								:= 		STRING_TO_INT(sProdCodeEK1110_End4);

//In this function block the CRC counts for the individual counts can be decoded
fbEK1110_EcGetSlaveCrcErrorEx(	
							sNetId					:= 		gc_sADSNetID,
							nSlaveAddr				:= 		gc_uiEK1110_EtherCATAdr,
							bExecute				:= 		xExecute,
							tTimeout				:= 		T#2S,
							bBusy					=> 		xEK1110GetSlaveCrc_Busy,
							bError					=> 		xEK1110GetSlaveCrc_Error,
							nErrId					=> 		udiEK1110GetSlaveCrc_ErrId,
							crcError				=> 		g_stHMI_EK1110CrcErrorEx );

//Working Counter: Should remain Zero, If value=1 then data is bad from this device
g_xEK1110_Wc ;


//Get the STATE of the AX5000 terminal and display as a text string
g_sHMI_StateAX5000 									:= 		F_ConvStateToString(g_wStateAX5000);

// slave device's STATE BITS  
g_stHMI_AX5000EcSlaveStateBits 						:=  	F_ConvSlaveStateToBits(g_stAX5000EcSlaveState);

fbAX5000_EcGetSlaveIdentity(		
							sNetId					:= 		gc_sADSNetID,
							nSlaveAddr				:= 		gc_uiAX5206_EtherCATAdr,
							bExecute				:= 		xExecute,
							tTimeout				:= 		T#2S,
							bBusy					=> 		xAX5000SlaveIdentity_Busy,
							bError					=> 		xAX5000SlaveIdentity_Error,
							nErrId					=> 		udiAX5000SlaveIdentity_ErrId,
							identity				=> 		stSlaveIdentityAX5000 );

sProdCodeAX5000 									:= 		F_ConvProductCodeToString(stSlaveIdentityAX5000);
//Get last 4 characters of the string
sProdCodeAX5000_End4 								:= 		RIGHT(sProdCodeAX5000, 4) ;
//Convert last 4 characters to a number
g_iHMI_ProdCodeAX5000 								:= 		STRING_TO_INT(sProdCodeAX5000_End4);

//In this function block the CRC counts for the individual counts can be decoded
fbAX5000_EcGetSlaveCrcErrorEx(	
							sNetId					:= 		gc_sADSNetID,
							nSlaveAddr				:= 		gc_uiAX5206_EtherCATAdr,
							bExecute				:= 		xExecute,
							tTimeout				:= 		T#2S,
							bBusy					=> 		xAX5000GetSlaveCrc_Busy,
							bError					=> 		xAX5000GetSlaveCrc_Error,
							nErrId					=> 		udiAX5000GetSlaveCrc_ErrId,
							crcError				=> 		g_stHMI_AX5000CrcErrorEx );

//Working Counter: Should remain Zero, If value=1 then data is bad from this device
g_xAX5000_Wc ;


//Get the STATE of the AX5805 terminal and display as a text string
g_sHMI_StateAX5805 									:= 		F_ConvStateToString(g_wStateAX5805);

// slave device's STATE BITS  
g_stHMI_AX5805EcSlaveStateBits 						:=  	F_ConvSlaveStateToBits(g_stAX5805EcSlaveState);

fbAX5805_EcGetSlaveIdentity(		
							sNetId					:= 		gc_sADSNetID,
							nSlaveAddr				:= 		gc_uiAX5805_EtherCATAdr,
							bExecute				:= 		xExecute,
							tTimeout				:= 		T#2S,
							bBusy					=> 		xAX5805SlaveIdentity_Busy,
							bError					=> 		xAX5805SlaveIdentity_Error,
							nErrId					=> 		udiAX5805SlaveIdentity_ErrId,
							identity				=> 		stSlaveIdentityAX5805 );

sProdCodeAX5805 									:= 		F_ConvProductCodeToString(stSlaveIdentityAX5805);
//Get last 4 characters of the string
sProdCodeAX5805_End4 								:= 		RIGHT(sProdCodeAX5805, 4) ;
//Convert last 4 characters to a number
g_iHMI_ProdCodeAX5805 								:= 		STRING_TO_INT(sProdCodeAX5805_End4);

//In this function block the CRC counts for the individual counts can be decoded
fbAX5805_EcGetSlaveCrcErrorEx(	
							sNetId					:= 		gc_sADSNetID,
							nSlaveAddr				:= 		gc_uiAX5805_EtherCATAdr,
							bExecute				:= 		xExecute,
							tTimeout				:= 		T#2S,
							bBusy					=> 		xAX5805GetSlaveCrc_Busy,
							bError					=> 		xAX5805GetSlaveCrc_Error,
							nErrId					=> 		udiAX5805GetSlaveCrc_ErrId,
							crcError				=> 		g_stHMI_AX5805CrcErrorEx );

//Working Counter: Should remain Zero, If value=1 then data is bad from this device
g_xAX5805_Wc ;


//Get the STATE of the EP1908-0002 module and display as a text string
g_sHMI_StateEP1908 									:= 		F_ConvStateToString(g_wStateEP1908);

// slave device's STATE BITS  
g_stHMI_EP1908EcSlaveStateBits 						:=  	F_ConvSlaveStateToBits(g_stEP1908EcSlaveState);

fbEP1908_EcGetSlaveIdentity(		
							sNetId					:= 		gc_sADSNetID,
							nSlaveAddr				:= 		gc_uiEP1908_EtherCATAdr,
							bExecute				:= 		xExecute,
							tTimeout				:= 		T#2S,
							bBusy					=> 		xEP1908SlaveIdentity_Busy,
							bError					=> 		xEP1908SlaveIdentity_Error,
							nErrId					=> 		udiEP1908SlaveIdentity_ErrId,
							identity				=> 		stSlaveIdentityEP1908 );

sProdCodeEP1908 									:= 		F_ConvProductCodeToString(stSlaveIdentityEP1908);
//Get last 4 characters of the string
sProdCodeEP1908_End4 								:= 		RIGHT(sProdCodeEP1908, 4) ;
//Convert last 4 characters to a number
g_iHMI_ProdCodeEP1908 								:= 		STRING_TO_INT(sProdCodeEP1908_End4);

//In this function block the CRC counts for the individual counts can be decoded
fbEP1908_EcGetSlaveCrcErrorEx(	
							sNetId					:= 		gc_sADSNetID,
							nSlaveAddr				:= 		gc_uiEP1908_EtherCATAdr,
							bExecute				:= 		xExecute,
							tTimeout				:= 		T#2S,
							bBusy					=> 		xEP1908GetSlaveCrc_Busy,
							bError					=> 		xEP1908GetSlaveCrc_Error,
							nErrId					=> 		udiEP1908GetSlaveCrc_ErrId,
							crcError				=> 		g_stHMI_EP1908CrcErrorEx );

